LIN {X 0,Y 467.683,Z 145.229,A -85,B 0,C 180,E1 -7462.66,E2 -7462.66} C_VEL
LIN {X 0,Y 467.713,Z 145.224,A -85,B 0,C 180,E1 -7464.827,E2 -7464.827} C_VEL
LIN {X 0,Y 467.852,Z 145.203,A -85,B 0,C 180,E1 -7467.417,E2 -7467.417} C_VEL
LIN {X 0,Y 467.855,Z 145.206,A -85,B 0,C 180,E1 -7470,E2 -7470} C_VEL
LIN {X 0,Y 467.817,Z 145.212,A -85,B 0,C 180,E1 -7472.583,E2 -7472.583} C_VEL
LIN {X 0,Y 467.706,Z 145.226,A -85,B 0,C 180,E1 -7476.038,E2 -7476.038} C_VEL
LIN {X 0,Y 467.661,Z 145.229,A -85,B 0,C 180,E1 -7478.643,E2 -7478.643} C_VEL
LIN {X 0,Y 467.66,Z 145.234,A -85,B 0,C 180,E1 -7482.145,E2 -7482.145} C_VEL
LIN {X 0,Y 467.615,Z 145.236,A -85,B 0,C 180,E1 -7485.696,E2 -7485.696} C_VEL
LIN {X 0,Y 467.621,Z 145.233,A -85,B 0,C 180,E1 -7489.308,E2 -7489.308} C_VEL
LIN {X 0,Y 467.536,Z 145.247,A -85,B 0,C 180,E1 -7492.074,E2 -7492.074} C_VEL
LIN {X 0,Y 467.562,Z 145.239,A -85,B 0,C 180,E1 -7494.89,E2 -7494.89} C_VEL
LIN {X 0,Y 467.548,Z 145.248,A -85,B 0,C 180,E1 -7497.774,E2 -7497.774} C_VEL
LIN {X 0,Y 467.568,Z 145.24,A -85,B 0,C 180,E1 -7501.044,E2 -7501.044} C_VEL
LIN {X 0,Y 467.579,Z 145.238,A -85,B 0,C 180,E1 -7504.24,E2 -7504.24} C_VEL
LIN {X 0,Y 467.545,Z 145.245,A -85,B 0,C 180,E1 -7507.185,E2 -7507.185} C_VEL
LIN {X 0,Y 467.56,Z 145.239,A -85,B 0,C 180,E1 -7510.267,E2 -7510.267} C_VEL
LIN {X 0,Y 467.547,Z 145.243,A -85,B 0,C 180,E1 -7513.746,E2 -7513.746} C_VEL
LIN {X 0,Y 467.547,Z 145.241,A -85,B 0,C 180,E1 -7516.254,E2 -7516.254} C_VEL
LIN {X 0,Y 467.56,Z 145.241,A -85,B 0,C 180,E1 -7519.733,E2 -7519.733} C_VEL
LIN {X 0,Y 467.546,Z 145.245,A -85,B 0,C 180,E1 -7522.815,E2 -7522.815} C_VEL
LIN {X 0,Y 467.579,Z 145.237,A -85,B 0,C 180,E1 -7525.76,E2 -7525.76} C_VEL
LIN {X 0,Y 467.546,Z 145.249,A -85,B 0,C 180,E1 -7528.961,E2 -7528.961} C_VEL
LIN {X 0,Y 467.563,Z 145.24,A -85,B 0,C 180,E1 -7532.227,E2 -7532.227} C_VEL
LIN {X 0,Y 467.563,Z 145.243,A -85,B 0,C 180,E1 -7535.11,E2 -7535.11} C_VEL
LIN {X 0,Y 467.529,Z 145.243,A -85,B 0,C 180,E1 -7537.926,E2 -7537.926} C_VEL
LIN {X 0,Y 467.62,Z 145.24,A -85,B 0,C 180,E1 -7540.692,E2 -7540.692} C_VEL
LIN {X 0,Y 467.616,Z 145.237,A -85,B 0,C 180,E1 -7544.304,E2 -7544.304} C_VEL
LIN {X 0,Y 467.661,Z 145.228,A -85,B 0,C 180,E1 -7547.855,E2 -7547.855} C_VEL
LIN {X 0,Y 467.639,Z 145.229,A -85,B 0,C 180,E1 -7551.356,E2 -7551.356} C_VEL
LIN {X 0,Y 467.705,Z 145.224,A -85,B 0,C 180,E1 -7553.962,E2 -7553.962} C_VEL
LIN {X 0,Y 467.816,Z 145.207,A -85,B 0,C 180,E1 -7557.417,E2 -7557.417} C_VEL
LIN {X 0,Y 467.853,Z 145.208,A -85,B 0,C 180,E1 -7560,E2 -7560} C_VEL
LIN {X 0,Y 467.815,Z 145.21,A -85,B 0,C 180,E1 -7562.583,E2 -7562.583} C_VEL
LIN {X 0,Y 467.704,Z 145.23,A -85,B 0,C 180,E1 -7566.038,E2 -7566.038} C_VEL
LIN {X 0,Y 467.637,Z 145.23,A -85,B 0,C 180,E1 -7568.644,E2 -7568.644} C_VEL
LIN {X 0,Y 467.652,Z 145.23,A -85,B 0,C 180,E1 -7572.354,E2 -7572.354} C_VEL
LIN {X 0,Y 467.574,Z 145.245,A -85,B 0,C 180,E1 -7575.851,E2 -7575.851} C_VEL
LIN {X 0,Y 467.571,Z 145.238,A -85,B 0,C 180,E1 -7578.746,E2 -7578.746} C_VEL
LIN {X 0,Y 467.521,Z 145.247,A -85,B 0,C 180,E1 -7582.075,E2 -7582.075} C_VEL
LIN {X 0,Y 467.553,Z 145.241,A -85,B 0,C 180,E1 -7584.89,E2 -7584.89} C_VEL
LIN {X 0,Y 467.54,Z 145.246,A -85,B 0,C 180,E1 -7587.774,E2 -7587.774} C_VEL
LIN {X 0,Y 467.53,Z 145.246,A -85,B 0,C 180,E1 -7591.036,E2 -7591.036} C_VEL
LIN {X 0,Y 467.567,Z 145.238,A -85,B 0,C 180,E1 -7594.237,E2 -7594.237} C_VEL
LIN {X 0,Y 467.516,Z 145.251,A -85,B 0,C 180,E1 -7597.18,E2 -7597.18} C_VEL
LIN {X 0,Y 467.553,Z 145.24,A -85,B 0,C 180,E1 -7600.267,E2 -7600.267} C_VEL
LIN {X 0,Y 467.519,Z 145.246,A -85,B 0,C 180,E1 -7602.568,E2 -7602.568} C_VEL
LIN {X 0,Y 467.564,Z 145.246,A -85,B 0,C 180,E1 -7605.052,E2 -7605.052} C_VEL
LIN {X 0,Y 467.556,Z 145.244,A -85,B 0,C 180,E1 -7608.727,E2 -7608.727} C_VEL
LIN {X 0,Y 467.539,Z 145.242,A -85,B 0,C 180,E1 -7611.953,E2 -7611.953} C_VEL
LIN {X 0,Y 467.542,Z 145.245,A -85,B 0,C 180,E1 -7615.165,E2 -7615.165} C_VEL
LIN {X 0,Y 467.544,Z 145.243,A -85,B 0,C 180,E1 -7618.257,E2 -7618.257} C_VEL
LIN {X 0,Y 467.526,Z 145.248,A -85,B 0,C 180,E1 -7621.247,E2 -7621.247} C_VEL
LIN {X 0,Y 467.561,Z 145.405,A -85,B 0,C 180,E1 -7624.405,E2 -7624.405} C_VEL
LIN {X 0,Y 469.547,Z 155.588,A -85,B 0,C 180,E1 -7626.398,E2 -7626.398} C_VEL
LIN {X 0,Y 469.65,Z 160.677,A -85,B 0,C 180,E1 -7627.335,E2 -7627.335} C_VEL
LIN {X 0,Y 468.851,Z 179.686,A -85,B 0,C 180,E1 -7630.745,E2 -7630.745} C_VEL
LIN {X 0,Y 468.323,Z 192.549,A -85,B 0,C 180,E1 -7633.009,E2 -7633.009} C_VEL
LIN {X 0,Y 471.154,Z 211.602,A -85,B 0,C 180,E1 -7633.413,E2 -7633.413} C_VEL
LIN {X 0,Y 470.437,Z 300.664,A -85,B 0,C 180,E1 -7634.817,E2 -7634.817} C_VEL
LIN {X 0,Y 470.098,Z 313.865,A -85,B 0,C 180,E1 -7635.194,E2 -7635.194} C_VEL
LIN {X 0,Y 469.617,Z 327.128,A -85,B 0,C 180,E1 -7635.759,E2 -7635.759} C_VEL
LIN {X 0,Y 469.107,Z 339.07,A -85,B 0,C 180,E1 -7636.462,E2 -7636.462} C_VEL
LIN {X 0,Y 468.56,Z 351.287,A -85,B 0,C 180,E1 -7637.392,E2 -7637.392} C_VEL
LIN {X 0,Y 468.159,Z 360.871,A -85,B 0,C 180,E1 -7638.307,E2 -7638.307} C_VEL
LIN {X 0,Y 467.696,Z 370.148,A -85,B 0,C 180,E1 -7639.392,E2 -7639.392} C_VEL
LIN {X 0,Y 467.304,Z 379.162,A -85,B 0,C 180,E1 -7640.696,E2 -7640.696} C_VEL
LIN {X 0,Y 467.007,Z 386.421,A -85,B 0,C 180,E1 -7641.998,E2 -7641.998} C_VEL
LIN {X 0,Y 466.833,Z 391.319,A -85,B 0,C 180,E1 -7643.083,E2 -7643.083} C_VEL
LIN {X 0,Y 466.755,Z 396.078,A -85,B 0,C 180,E1 -7644.383,E2 -7644.383} C_VEL
LIN {X 0,Y 466.645,Z 399.712,A -85,B 0,C 180,E1 -7645.681,E2 -7645.681} C_VEL
LIN {X 0,Y 466.688,Z 401.59,A -85,B 0,C 180,E1 -7646.547,E2 -7646.547} C_VEL
LIN {X 0,Y 466.662,Z 402.997,A -85,B 0,C 180,E1 -7647.41,E2 -7647.41} C_VEL
LIN {X 0,Y 466.62,Z 404.607,A -85,B 0,C 180,E1 -7649.137,E2 -7649.137} C_VEL
LIN {X 0,Y 466.601,Z 404.824,A -85,B 0,C 180,E1 -7650,E2 -7650} C_VEL
LIN {X 0,Y 466.62,Z 404.607,A -85,B 0,C 180,E1 -7650.863,E2 -7650.863} C_VEL
LIN {X 0,Y 466.662,Z 402.991,A -85,B 0,C 180,E1 -7652.59,E2 -7652.59} C_VEL
LIN {X 0,Y 466.688,Z 401.586,A -85,B 0,C 180,E1 -7653.453,E2 -7653.453} C_VEL
LIN {X 0,Y 466.687,Z 398.63,A -85,B 0,C 180,E1 -7654.751,E2 -7654.751} C_VEL
LIN {X 0,Y 466.744,Z 394.631,A -85,B 0,C 180,E1 -7656.05,E2 -7656.05} C_VEL
LIN {X 0,Y 466.94,Z 388.484,A -85,B 0,C 180,E1 -7657.568,E2 -7657.568} C_VEL
LIN {X 0,Y 467.199,Z 381.769,A -85,B 0,C 180,E1 -7658.87,E2 -7658.87} C_VEL
LIN {X 0,Y 467.53,Z 373.439,A -85,B 0,C 180,E1 -7660.174,E2 -7660.174} C_VEL
LIN {X 0,Y 467.998,Z 364.898,A -85,B 0,C 180,E1 -7661.258,E2 -7661.258} C_VEL
LIN {X 0,Y 468.486,Z 354.809,A -85,B 0,C 180,E1 -7662.301,E2 -7662.301} C_VEL
LIN {X 0,Y 468.939,Z 343.914,A -85,B 0,C 180,E1 -7663.212,E2 -7663.212} C_VEL
LIN {X 0,Y 469.412,Z 332.466,A -85,B 0,C 180,E1 -7663.971,E2 -7663.971} C_VEL
LIN {X 0,Y 469.895,Z 320.661,A -85,B 0,C 180,E1 -7664.564,E2 -7664.564} C_VEL
LIN {X 0,Y 470.317,Z 307.075,A -85,B 0,C 180,E1 -7665.049,E2 -7665.049} C_VEL
LIN {X 0,Y 470.645,Z 293.364,A -85,B 0,C 180,E1 -7665.343,E2 -7665.343} C_VEL
LIN {X 0,Y 471.151,Z 210.06,A -85,B 0,C 180,E1 -7666.648,E2 -7666.648} C_VEL
LIN {X 0,Y 468.307,Z 191.951,A -85,B 0,C 180,E1 -7667.066,E2 -7667.066} C_VEL
LIN {X 0,Y 468.86,Z 176.916,A -85,B 0,C 180,E1 -7669.711,E2 -7669.711} C_VEL
LIN {X 0,Y 469.689,Z 159.022,A -85,B 0,C 180,E1 -7672.895,E2 -7672.895} C_VEL
LIN {X 0,Y 469.27,Z 153.888,A -85,B 0,C 180,E1 -7673.852,E2 -7673.852} C_VEL
LIN {X 0,Y 467.557,Z 145.248,A -85,B 0,C 180,E1 -7675.544,E2 -7675.544} C_VEL
LIN {X 0,Y 467.526,Z 145.25,A -85,B 0,C 180,E1 -7678.753,E2 -7678.753} C_VEL
LIN {X 0,Y 467.544,Z 145.249,A -85,B 0,C 180,E1 -7681.743,E2 -7681.743} C_VEL
LIN {X 0,Y 467.541,Z 145.248,A -85,B 0,C 180,E1 -7684.835,E2 -7684.835} C_VEL
LIN {X 0,Y 467.535,Z 145.244,A -85,B 0,C 180,E1 -7688.048,E2 -7688.048} C_VEL
LIN {X 0,Y 467.551,Z 145.245,A -85,B 0,C 180,E1 -7691.406,E2 -7691.406} C_VEL
LIN {X 0,Y 467.564,Z 145.247,A -85,B 0,C 180,E1 -7695.052,E2 -7695.052} C_VEL
LIN {X 0,Y 467.552,Z 145.246,A -85,B 0,C 180,E1 -7698.728,E2 -7698.728} C_VEL
LIN {X 0,Y 467.536,Z 145.243,A -85,B 0,C 180,E1 -7701.953,E2 -7701.953} C_VEL
LIN {X 0,Y 467.543,Z 145.245,A -85,B 0,C 180,E1 -7705.165,E2 -7705.165} C_VEL
LIN {X 0,Y 467.545,Z 145.242,A -85,B 0,C 180,E1 -7708.257,E2 -7708.257} C_VEL
LIN {X 0,Y 467.527,Z 145.243,A -85,B 0,C 180,E1 -7711.247,E2 -7711.247} C_VEL
LIN {X 0,Y 467.564,Z 145.243,A -85,B 0,C 180,E1 -7714.406,E2 -7714.406} C_VEL
LIN {X 0,Y 467.549,Z 145.244,A -85,B 0,C 180,E1 -7716.994,E2 -7716.994} C_VEL
LIN {X 0,Y 467.541,Z 145.237,A -85,B 0,C 180,E1 -7719.773,E2 -7719.773} C_VEL
LIN {X 0,Y 467.555,Z 145.246,A -85,B 0,C 180,E1 -7722.505,E2 -7722.505} C_VEL
LIN {X 0,Y 467.562,Z 145.238,A -85,B 0,C 180,E1 -7725.195,E2 -7725.195} C_VEL
LIN {X 0,Y 467.645,Z 145.23,A -85,B 0,C 180,E1 -7727.854,E2 -7727.854} C_VEL
LIN {X 0,Y 467.633,Z 145.23,A -85,B 0,C 180,E1 -7731.356,E2 -7731.356} C_VEL
LIN {X 0,Y 467.697,Z 145.221,A -85,B 0,C 180,E1 -7733.962,E2 -7733.962} C_VEL
LIN {X 0,Y 467.815,Z 145.205,A -85,B 0,C 180,E1 -7737.417,E2 -7737.417} C_VEL
LIN {X 0,Y 467.853,Z 145.208,A -85,B 0,C 180,E1 -7740,E2 -7740} C_VEL
LIN {X 0,Y 467.815,Z 145.209,A -85,B 0,C 180,E1 -7742.583,E2 -7742.583} C_VEL
LIN {X 0,Y 467.704,Z 145.225,A -85,B 0,C 180,E1 -7746.038,E2 -7746.038} C_VEL
LIN {X 0,Y 467.637,Z 145.23,A -85,B 0,C 180,E1 -7748.644,E2 -7748.644} C_VEL
LIN {X 0,Y 467.652,Z 145.231,A -85,B 0,C 180,E1 -7752.146,E2 -7752.146} C_VEL
LIN {X 0,Y 467.617,Z 145.237,A -85,B 0,C 180,E1 -7755.696,E2 -7755.696} C_VEL
LIN {X 0,Y 467.576,Z 145.238,A -85,B 0,C 180,E1 -7758.748,E2 -7758.748} C_VEL
LIN {X 0,Y 467.562,Z 145.242,A -85,B 0,C 180,E1 -7761.261,E2 -7761.261} C_VEL
LIN {X 0,Y 467.558,Z 145.246,A -85,B 0,C 180,E1 -7763.944,E2 -7763.944} C_VEL
LIN {X 0,Y 467.538,Z 145.246,A -85,B 0,C 180,E1 -7766.805,E2 -7766.805} C_VEL
LIN {X 0,Y 467.538,Z 145.249,A -85,B 0,C 180,E1 -7769.739,E2 -7769.739} C_VEL
LIN {X 0,Y 467.577,Z 145.242,A -85,B 0,C 180,E1 -7772.759,E2 -7772.759} C_VEL
LIN {X 0,Y 467.567,Z 145.246,A -85,B 0,C 180,E1 -7775.889,E2 -7775.889} C_VEL
LIN {X 0,Y 467.613,Z 145.348,A -85,B 0,C 180,E1 -7776.318,E2 -7776.318} C_VEL
LIN {X 0,Y 468.909,Z 152.961,A -85,B 0,C 180,E1 -7777.916,E2 -7777.916} C_VEL
LIN {X 0,Y 468.662,Z 165.61,A -85,B 0,C 180,E1 -7780.434,E2 -7780.434} C_VEL
LIN {X 0,Y 468.541,Z 168.542,A -85,B 0,C 180,E1 -7781.014,E2 -7781.014} C_VEL
LIN {X 0,Y 471.427,Z 183.586,A -85,B 0,C 180,E1 -7781.373,E2 -7781.373} C_VEL
LIN {X 0,Y 470.577,Z 276.466,A -85,B 0,C 180,E1 -7782.849,E2 -7782.849} C_VEL
LIN {X 0,Y 470.298,Z 290.13,A -85,B 0,C 180,E1 -7783.255,E2 -7783.255} C_VEL
LIN {X 0,Y 469.95,Z 302.218,A -85,B 0,C 180,E1 -7783.785,E2 -7783.785} C_VEL
LIN {X 0,Y 469.476,Z 313.638,A -85,B 0,C 180,E1 -7784.456,E2 -7784.456} C_VEL
LIN {X 0,Y 468.981,Z 325.331,A -85,B 0,C 180,E1 -7785.343,E2 -7785.343} C_VEL
LIN {X 0,Y 468.475,Z 336.021,A -85,B 0,C 180,E1 -7786.363,E2 -7786.363} C_VEL
LIN {X 0,Y 467.997,Z 345.447,A -85,B 0,C 180,E1 -7787.485,E2 -7787.485} C_VEL
LIN {X 0,Y 467.583,Z 353.89,A -85,B 0,C 180,E1 -7788.723,E2 -7788.723} C_VEL
LIN {X 0,Y 467.232,Z 361.432,A -85,B 0,C 180,E1 -7790.097,E2 -7790.097} C_VEL
LIN {X 0,Y 466.981,Z 367.45,A -85,B 0,C 180,E1 -7791.499,E2 -7791.499} C_VEL
LIN {X 0,Y 466.806,Z 372.297,A -85,B 0,C 180,E1 -7792.971,E2 -7792.971} C_VEL
LIN {X 0,Y 466.634,Z 375.76,A -85,B 0,C 180,E1 -7794.42,E2 -7794.42} C_VEL
LIN {X 0,Y 466.534,Z 378.282,A -85,B 0,C 180,E1 -7796.125,E2 -7796.125} C_VEL
LIN {X 0,Y 466.51,Z 379.06,A -85,B 0,C 180,E1 -7797.217,E2 -7797.217} C_VEL
LIN {X 0,Y 465.851,Z 379.263,A -85,B 0,C 180,E1 -7797.938,E2 -7797.938} C_VEL
LIN {X 0,Y 463.014,Z 379.028,A -85,B 0,C 180,E1 -7799.111,E2 -7799.111} C_VEL
LIN {X 0,Y 460.619,Z 378.334,A -85,B 0,C 180,E1 -7800.053,E2 -7800.053} C_VEL
LIN {X 0,Y 459.537,Z 377.298,A -85,B 0,C 180,E1 -7800.894,E2 -7800.894} C_VEL
LIN {X 0,Y 459.517,Z 377.041,A -85,B 0,C 180,E1 -7801.015,E2 -7801.015} C_VEL
LIN {X 0,Y 459.644,Z 374.212,A -85,B 0,C 180,E1 -7802.478,E2 -7802.478} C_VEL
LIN {X 0,Y 459.894,Z 369.669,A -85,B 0,C 180,E1 -7804.067,E2 -7804.067} C_VEL
LIN {X 0,Y 460.064,Z 363.549,A -85,B 0,C 180,E1 -7805.641,E2 -7805.641} C_VEL
LIN {X 0,Y 460.415,Z 356.212,A -85,B 0,C 180,E1 -7807.092,E2 -7807.092} C_VEL
LIN {X 0,Y 460.81,Z 348.502,A -85,B 0,C 180,E1 -7808.317,E2 -7808.317} C_VEL
LIN {X 0,Y 461.276,Z 339.442,A -85,B 0,C 180,E1 -7809.486,E2 -7809.486} C_VEL
LIN {X 0,Y 461.796,Z 328.795,A -85,B 0,C 180,E1 -7810.592,E2 -7810.592} C_VEL
LIN {X 0,Y 462.388,Z 317.849,A -85,B 0,C 180,E1 -7811.501,E2 -7811.501} C_VEL
LIN {X 0,Y 462.805,Z 306.173,A -85,B 0,C 180,E1 -7812.262,E2 -7812.262} C_VEL
LIN {X 0,Y 463.234,Z 292.993,A -85,B 0,C 180,E1 -7812.904,E2 -7812.904} C_VEL
LIN {X 0,Y 463.559,Z 280.962,A -85,B 0,C 180,E1 -7813.315,E2 -7813.315} C_VEL
LIN {X 0,Y 463.764,Z 266.671,A -85,B 0,C 180,E1 -7813.605,E2 -7813.605} C_VEL
LIN {X 0,Y 464.504,Z 184.737,A -85,B 0,C 180,E1 -7814.899,E2 -7814.899} C_VEL
LIN {X 0,Y 461.504,Z 168.599,A -85,B 0,C 180,E1 -7815.278,E2 -7815.278} C_VEL
LIN {X 0,Y 461.992,Z 154.759,A -85,B 0,C 180,E1 -7818.149,E2 -7818.149} C_VEL
LIN {X 0,Y 460.626,Z 146.11,A -85,B 0,C 180,E1 -7820.061,E2 -7820.061} C_VEL
LIN {X 0,Y 460.612,Z 146.111,A -85,B 0,C 180,E1 -7822.989,E2 -7822.989} C_VEL
LIN {X 0,Y 460.685,Z 146.1,A -85,B 0,C 180,E1 -7824.748,E2 -7824.748} C_VEL
LIN {X 0,Y 460.792,Z 146.082,A -85,B 0,C 180,E1 -7827.377,E2 -7827.377} C_VEL
LIN {X 0,Y 460.825,Z 146.081,A -85,B 0,C 180,E1 -7830,E2 -7830} C_VEL
LIN {X 0,Y 460.761,Z 146.09,A -85,B 0,C 180,E1 -7832.623,E2 -7832.623} C_VEL
LIN {X 0,Y 460.672,Z 146.104,A -85,B 0,C 180,E1 -7836.13,E2 -7836.13} C_VEL
LIN {X 0,Y 460.613,Z 146.106,A -85,B 0,C 180,E1 -7838.776,E2 -7838.776} C_VEL
LIN {X 0,Y 460.612,Z 146.109,A -85,B 0,C 180,E1 -7842.334,E2 -7842.334} C_VEL
LIN {X 0,Y 460.559,Z 146.119,A -85,B 0,C 180,E1 -7845.978,E2 -7845.978} C_VEL
LIN {X 0,Y 460.568,Z 146.114,A -85,B 0,C 180,E1 -7849.616,E2 -7849.616} C_VEL
LIN {X 0,Y 460.513,Z 146.118,A -85,B 0,C 180,E1 -7852.429,E2 -7852.429} C_VEL
LIN {X 0,Y 460.537,Z 146.122,A -85,B 0,C 180,E1 -7855.793,E2 -7855.793} C_VEL
LIN {X 0,Y 460.523,Z 146.118,A -85,B 0,C 180,E1 -7859.232,E2 -7859.232} C_VEL
LIN {X 0,Y 460.528,Z 146.116,A -85,B 0,C 180,E1 -7862.285,E2 -7862.285} C_VEL
LIN {X 0,Y 460.509,Z 146.125,A -85,B 0,C 180,E1 -7865.446,E2 -7865.446} C_VEL
LIN {X 0,Y 460.507,Z 146.12,A -85,B 0,C 180,E1 -7868.891,E2 -7868.891} C_VEL
LIN {X 0,Y 460.505,Z 146.123,A -85,B 0,C 180,E1 -7871.598,E2 -7871.598} C_VEL
LIN {X 0,Y 460.514,Z 146.118,A -85,B 0,C 180,E1 -7874.589,E2 -7874.589} C_VEL
LIN {X 0,Y 460.478,Z 146.123,A -85,B 0,C 180,E1 -7877.813,E2 -7877.813} C_VEL
LIN {X 0,Y 460.516,Z 146.117,A -85,B 0,C 180,E1 -7880.136,E2 -7880.136} C_VEL
LIN {X 0,Y 460.476,Z 146.125,A -85,B 0,C 180,E1 -7883.47,E2 -7883.47} C_VEL
LIN {X 0,Y 460.519,Z 146.12,A -85,B 0,C 180,E1 -7886.674,E2 -7886.674} C_VEL
LIN {X 0,Y 460.5,Z 146.119,A -85,B 0,C 180,E1 -7889.759,E2 -7889.759} C_VEL
LIN {X 0,Y 460.516,Z 146.123,A -85,B 0,C 180,E1 -7892.752,E2 -7892.752} C_VEL
LIN {X 0,Y 460.521,Z 146.116,A -85,B 0,C 180,E1 -7895.666,E2 -7895.666} C_VEL
LIN {X 0,Y 460.522,Z 146.122,A -85,B 0,C 180,E1 -7898.58,E2 -7898.58} C_VEL
LIN {X 0,Y 460.586,Z 146.109,A -85,B 0,C 180,E1 -7901.311,E2 -7901.311} C_VEL
LIN {X 0,Y 460.549,Z 146.115,A -85,B 0,C 180,E1 -7904.964,E2 -7904.964} C_VEL
LIN {X 0,Y 460.613,Z 146.111,A -85,B 0,C 180,E1 -7908.559,E2 -7908.559} C_VEL
LIN {X 0,Y 460.597,Z 146.107,A -85,B 0,C 180,E1 -7911.223,E2 -7911.223} C_VEL
LIN {X 0,Y 460.671,Z 146.1,A -85,B 0,C 180,E1 -7913.87,E2 -7913.87} C_VEL
LIN {X 0,Y 460.76,Z 146.086,A -85,B 0,C 180,E1 -7917.377,E2 -7917.377} C_VEL
LIN {X 0,Y 460.823,Z 146.084,A -85,B 0,C 180,E1 -7920,E2 -7920} C_VEL
LIN {X 0,Y 460.759,Z 146.088,A -85,B 0,C 180,E1 -7922.623,E2 -7922.623} C_VEL
LIN {X 0,Y 460.67,Z 146.104,A -85,B 0,C 180,E1 -7926.13,E2 -7926.13} C_VEL
LIN {X 0,Y 460.592,Z 146.108,A -85,B 0,C 180,E1 -7928.777,E2 -7928.777} C_VEL
LIN {X 0,Y 460.601,Z 146.108,A -85,B 0,C 180,E1 -7932.435,E2 -7932.435} C_VEL
LIN {X 0,Y 460.529,Z 146.121,A -85,B 0,C 180,E1 -7935.964,E2 -7935.964} C_VEL
LIN {X 0,Y 460.53,Z 146.115,A -85,B 0,C 180,E1 -7938.885,E2 -7938.885} C_VEL
LIN {X 0,Y 460.495,Z 146.12,A -85,B 0,C 180,E1 -7942.43,E2 -7942.43} C_VEL
LIN {X 0,Y 460.524,Z 146.121,A -85,B 0,C 180,E1 -7945.789,E2 -7945.789} C_VEL
LIN {X 0,Y 460.498,Z 146.119,A -85,B 0,C 180,E1 -7948.237,E2 -7948.237} C_VEL
LIN {X 0,Y 460.498,Z 146.125,A -85,B 0,C 180,E1 -7951.277,E2 -7951.277} C_VEL
LIN {X 0,Y 460.513,Z 146.117,A -85,B 0,C 180,E1 -7954.501,E2 -7954.501} C_VEL
LIN {X 0,Y 460.483,Z 146.124,A -85,B 0,C 180,E1 -7957.625,E2 -7957.625} C_VEL
LIN {X 0,Y 460.515,Z 146.122,A -85,B 0,C 180,E1 -7961.013,E2 -7961.013} C_VEL
LIN {X 0,Y 460.512,Z 146.119,A -85,B 0,C 180,E1 -7964.589,E2 -7964.589} C_VEL
LIN {X 0,Y 460.474,Z 146.122,A -85,B 0,C 180,E1 -7967.813,E2 -7967.813} C_VEL
LIN {X 0,Y 460.497,Z 146.119,A -85,B 0,C 180,E1 -7970.134,E2 -7970.134} C_VEL
LIN {X 0,Y 460.458,Z 146.125,A -85,B 0,C 180,E1 -7973.469,E2 -7973.469} C_VEL
LIN {X 0,Y 460.501,Z 146.125,A -85,B 0,C 180,E1 -7976.673,E2 -7976.673} C_VEL
LIN {X 0,Y 460.479,Z 146.124,A -85,B 0,C 180,E1 -7979.757,E2 -7979.757} C_VEL
LIN {X 0,Y 460.485,Z 146.128,A -85,B 0,C 180,E1 -7982.75,E2 -7982.75} C_VEL
LIN {X 0,Y 460.546,Z 146.304,A -85,B 0,C 180,E1 -7984.204,E2 -7984.204} C_VEL
LIN {X 0,Y 462.709,Z 157.916,A -85,B 0,C 180,E1 -7986.504,E2 -7986.504} C_VEL
LIN {X 0,Y 462.351,Z 169.326,A -85,B 0,C 180,E1 -7988.604,E2 -7988.604} C_VEL
LIN {X 0,Y 461.645,Z 184.525,A -85,B 0,C 180,E1 -7991.355,E2 -7991.355} C_VEL
LIN {X 0,Y 461.351,Z 192.266,A -85,B 0,C 180,E1 -7992.746,E2 -7992.746} C_VEL
LIN {X 0,Y 464.335,Z 211.934,A -85,B 0,C 180,E1 -7993.178,E2 -7993.178} C_VEL
LIN {X 0,Y 463.596,Z 300.067,A -85,B 0,C 180,E1 -7994.587,E2 -7994.587} C_VEL
LIN {X 0,Y 463.226,Z 313.409,A -85,B 0,C 180,E1 -7994.969,E2 -7994.969} C_VEL
LIN {X 0,Y 462.738,Z 326.75,A -85,B 0,C 180,E1 -7995.543,E2 -7995.543} C_VEL
LIN {X 0,Y 462.181,Z 338.745,A -85,B 0,C 180,E1 -7996.255,E2 -7996.255} C_VEL
LIN {X 0,Y 461.65,Z 350.343,A -85,B 0,C 180,E1 -7997.145,E2 -7997.145} C_VEL
LIN {X 0,Y 461.19,Z 360.599,A -85,B 0,C 180,E1 -7998.128,E2 -7998.128} C_VEL
LIN {X 0,Y 460.662,Z 369.896,A -85,B 0,C 180,E1 -7999.229,E2 -7999.229} C_VEL
LIN {X 0,Y 460.258,Z 378.924,A -85,B 0,C 180,E1 -8000.552,E2 -8000.552} C_VEL
LIN {X 0,Y 459.948,Z 386.193,A -85,B 0,C 180,E1 -8001.875,E2 -8001.875} C_VEL
LIN {X 0,Y 459.737,Z 392.286,A -85,B 0,C 180,E1 -8003.272,E2 -8003.272} C_VEL
LIN {X 0,Y 459.647,Z 397.193,A -85,B 0,C 180,E1 -8004.736,E2 -8004.736} C_VEL
LIN {X 0,Y 459.563,Z 399.505,A -85,B 0,C 180,E1 -8005.615,E2 -8005.615} C_VEL
LIN {X 0,Y 459.583,Z 401.385,A -85,B 0,C 180,E1 -8006.493,E2 -8006.493} C_VEL
LIN {X 0,Y 459.584,Z 402.797,A -85,B 0,C 180,E1 -8007.371,E2 -8007.371} C_VEL
LIN {X 0,Y 459.523,Z 404.41,A -85,B 0,C 180,E1 -8009.124,E2 -8009.124} C_VEL
LIN {X 0,Y 459.533,Z 404.63,A -85,B 0,C 180,E1 -8010,E2 -8010} C_VEL
LIN {X 0,Y 459.523,Z 404.414,A -85,B 0,C 180,E1 -8010.876,E2 -8010.876} C_VEL
LIN {X 0,Y 459.584,Z 402.8,A -85,B 0,C 180,E1 -8012.629,E2 -8012.629} C_VEL
LIN {X 0,Y 459.583,Z 401.395,A -85,B 0,C 180,E1 -8013.507,E2 -8013.507} C_VEL
LIN {X 0,Y 459.615,Z 398.44,A -85,B 0,C 180,E1 -8014.824,E2 -8014.824} C_VEL
LIN {X 0,Y 459.714,Z 393.408,A -85,B 0,C 180,E1 -8016.431,E2 -8016.431} C_VEL
LIN {X 0,Y 459.898,Z 387.282,A -85,B 0,C 180,E1 -8017.905,E2 -8017.905} C_VEL
LIN {X 0,Y 460.196,Z 380.345,A -85,B 0,C 180,E1 -8019.228,E2 -8019.228} C_VEL
LIN {X 0,Y 460.488,Z 373.262,A -85,B 0,C 180,E1 -8020.331,E2 -8020.331} C_VEL
LIN {X 0,Y 461.016,Z 364.728,A -85,B 0,C 180,E1 -8021.431,E2 -8021.431} C_VEL
LIN {X 0,Y 461.504,Z 354.852,A -85,B 0,C 180,E1 -8022.47,E2 -8022.47} C_VEL
LIN {X 0,Y 462.016,Z 343.755,A -85,B 0,C 180,E1 -8023.414,E2 -8023.414} C_VEL
LIN {X 0,Y 462.525,Z 332.32,A -85,B 0,C 180,E1 -8024.183,E2 -8024.183} C_VEL
LIN {X 0,Y 463.033,Z 320.547,A -85,B 0,C 180,E1 -8024.785,E2 -8024.785} C_VEL
LIN {X 0,Y 463.485,Z 307.01,A -85,B 0,C 180,E1 -8025.276,E2 -8025.276} C_VEL
LIN {X 0,Y 463.826,Z 293.453,A -85,B 0,C 180,E1 -8025.574,E2 -8025.574} C_VEL
LIN {X 0,Y 464.322,Z 210.557,A -85,B 0,C 180,E1 -8026.897,E2 -8026.897} C_VEL
LIN {X 0,Y 461.359,Z 191.816,A -85,B 0,C 180,E1 -8027.326,E2 -8027.326} C_VEL
LIN {X 0,Y 462.014,Z 175.48,A -85,B 0,C 180,E1 -8030.247,E2 -8030.247} C_VEL
LIN {X 0,Y 462.772,Z 158.873,A -85,B 0,C 180,E1 -8033.257,E2 -8033.257} C_VEL
LIN {X 0,Y 461.291,Z 149.874,A -85,B 0,C 180,E1 -8035.011,E2 -8035.011} C_VEL
LIN {X 0,Y 460.524,Z 146.122,A -85,B 0,C 180,E1 -8035.79,E2 -8035.79} C_VEL
LIN {X 0,Y 460.497,Z 146.125,A -85,B 0,C 180,E1 -8038.237,E2 -8038.237} C_VEL
LIN {X 0,Y 460.497,Z 146.129,A -85,B 0,C 180,E1 -8041.278,E2 -8041.278} C_VEL
LIN {X 0,Y 460.51,Z 146.122,A -85,B 0,C 180,E1 -8044.501,E2 -8044.501} C_VEL
LIN {X 0,Y 460.479,Z 146.125,A -85,B 0,C 180,E1 -8047.626,E2 -8047.626} C_VEL
LIN {X 0,Y 460.501,Z 146.128,A -85,B 0,C 180,E1 -8051.015,E2 -8051.015} C_VEL
LIN {X 0,Y 460.512,Z 146.122,A -85,B 0,C 180,E1 -8054.59,E2 -8054.59} C_VEL
LIN {X 0,Y 460.473,Z 146.124,A -85,B 0,C 180,E1 -8057.813,E2 -8057.813} C_VEL
LIN {X 0,Y 460.476,Z 146.121,A -85,B 0,C 180,E1 -8060.132,E2 -8060.132} C_VEL
LIN {X 0,Y 460.457,Z 146.124,A -85,B 0,C 180,E1 -8063.469,E2 -8063.469} C_VEL
LIN {X 0,Y 460.503,Z 146.122,A -85,B 0,C 180,E1 -8066.673,E2 -8066.673} C_VEL
LIN {X 0,Y 460.481,Z 146.121,A -85,B 0,C 180,E1 -8069.758,E2 -8069.758} C_VEL
LIN {X 0,Y 460.487,Z 146.127,A -85,B 0,C 180,E1 -8072.751,E2 -8072.751} C_VEL
LIN {X 0,Y 460.498,Z 146.116,A -85,B 0,C 180,E1 -8075.665,E2 -8075.665} C_VEL
LIN {X 0,Y 460.513,Z 146.12,A -85,B 0,C 180,E1 -8078.583,E2 -8078.583} C_VEL
LIN {X 0,Y 460.53,Z 146.116,A -85,B 0,C 180,E1 -8081.308,E2 -8081.308} C_VEL
LIN {X 0,Y 460.524,Z 146.117,A -85,B 0,C 180,E1 -8084.056,E2 -8084.056} C_VEL
LIN {X 0,Y 460.605,Z 146.106,A -85,B 0,C 180,E1 -8087.666,E2 -8087.666} C_VEL
LIN {X 0,Y 460.589,Z 146.107,A -85,B 0,C 180,E1 -8091.223,E2 -8091.223} C_VEL
LIN {X 0,Y 460.664,Z 146.096,A -85,B 0,C 180,E1 -8093.869,E2 -8093.869} C_VEL
LIN {X 0,Y 460.758,Z 146.084,A -85,B 0,C 180,E1 -8097.377,E2 -8097.377} C_VEL
LIN {X 0,Y 460.822,Z 146.084,A -85,B 0,C 180,E1 -8100,E2 -8100} C_VEL
LIN {X 0,Y 460.759,Z 146.088,A -85,B 0,C 180,E1 -8102.623,E2 -8102.623} C_VEL
LIN {X 0,Y 460.671,Z 146.101,A -85,B 0,C 180,E1 -8106.13,E2 -8106.13} C_VEL
LIN {X 0,Y 460.592,Z 146.107,A -85,B 0,C 180,E1 -8108.777,E2 -8108.777} C_VEL
LIN {X 0,Y 460.601,Z 146.107,A -85,B 0,C 180,E1 -8112.435,E2 -8112.435} C_VEL
LIN {X 0,Y 460.561,Z 146.117,A -85,B 0,C 180,E1 -8115.978,E2 -8115.978} C_VEL
LIN {X 0,Y 460.534,Z 146.115,A -85,B 0,C 180,E1 -8118.886,E2 -8118.886} C_VEL
LIN {X 0,Y 460.513,Z 146.123,A -85,B 0,C 180,E1 -8121.486,E2 -8121.486} C_VEL
LIN {X 0,Y 460.521,Z 146.12,A -85,B 0,C 180,E1 -8124.334,E2 -8124.334} C_VEL
LIN {X 0,Y 460.494,Z 146.127,A -85,B 0,C 180,E1 -8127.249,E2 -8127.249} C_VEL
LIN {X 0,Y 460.5,Z 146.123,A -85,B 0,C 180,E1 -8130.241,E2 -8130.241} C_VEL
LIN {X 0,Y 460.52,Z 146.123,A -85,B 0,C 180,E1 -8133.326,E2 -8133.326} C_VEL
LIN {X 0,Y 460.569,Z 146.269,A -85,B 0,C 180,E1 -8136.121,E2 -8136.121} C_VEL
LIN {X 0,Y 461.919,Z 153.671,A -85,B 0,C 180,E1 -8137.704,E2 -8137.704} C_VEL
LIN {X 0,Y 461.782,Z 163.71,A -85,B 0,C 180,E1 -8139.733,E2 -8139.733} C_VEL
LIN {X 0,Y 461.617,Z 168.827,A -85,B 0,C 180,E1 -8140.746,E2 -8140.746} C_VEL
LIN {X 0,Y 464.59,Z 183.936,A -85,B 0,C 180,E1 -8141.115,E2 -8141.115} C_VEL
LIN {X 0,Y 463.756,Z 276.622,A -85,B 0,C 180,E1 -8142.614,E2 -8142.614} C_VEL
LIN {X 0,Y 463.483,Z 290.022,A -85,B 0,C 180,E1 -8143.016,E2 -8143.016} C_VEL
LIN {X 0,Y 463.097,Z 302.314,A -85,B 0,C 180,E1 -8143.559,E2 -8143.559} C_VEL
LIN {X 0,Y 462.55,Z 314.455,A -85,B 0,C 180,E1 -8144.289,E2 -8144.289} C_VEL
LIN {X 0,Y 462.057,Z 325.458,A -85,B 0,C 180,E1 -8145.14,E2 -8145.14} C_VEL
LIN {X 0,Y 461.531,Z 335.875,A -85,B 0,C 180,E1 -8146.143,E2 -8146.143} C_VEL
LIN {X 0,Y 461.015,Z 345.372,A -85,B 0,C 180,E1 -8147.282,E2 -8147.282} C_VEL
LIN {X 0,Y 460.612,Z 352.934,A -85,B 0,C 180,E1 -8148.387,E2 -8148.387} C_VEL
LIN {X 0,Y 460.271,Z 360.631,A -85,B 0,C 180,E1 -8149.771,E2 -8149.771} C_VEL
LIN {X 0,Y 459.979,Z 366.977,A -85,B 0,C 180,E1 -8151.212,E2 -8151.212} C_VEL
LIN {X 0,Y 459.741,Z 371.82,A -85,B 0,C 180,E1 -8152.648,E2 -8152.648} C_VEL
LIN {X 0,Y 459.6,Z 375.512,A -85,B 0,C 180,E1 -8154.141,E2 -8154.141} C_VEL
LIN {X 0,Y 459.466,Z 378.03,A -85,B 0,C 180,E1 -8155.689,E2 -8155.689} C_VEL
LIN {X 0,Y 459.415,Z 379.312,A -85,B 0,C 180,E1 -8157.286,E2 -8157.286} C_VEL
LIN {X 0,Y 459.438,Z 379.209,A -85,B 0,C 180,E1 -8158.941,E2 -8158.941} C_VEL
LIN {X 0,Y 459.522,Z 377.571,A -85,B 0,C 180,E1 -8160.698,E2 -8160.698} C_VEL
LIN {X 0,Y 459.517,Z 377.041,A -85,B 0,C 180,E1 -8161.015,E2 -8161.015} C_VEL
LIN {X 0,Y 458.878,Z 375.872,A -85,B 0,C 180,E1 -8161.731,E2 -8161.731} C_VEL
LIN {X 0,Y 456.126,Z 373.403,A -85,B 0,C 180,E1 -8162.883,E2 -8162.883} C_VEL
LIN {X 0,Y 453.845,Z 370.936,A -85,B 0,C 180,E1 -8163.795,E2 -8163.795} C_VEL
LIN {X 0,Y 452.932,Z 368.729,A -85,B 0,C 180,E1 -8164.483,E2 -8164.483} C_VEL
LIN {X 0,Y 452.893,Z 367.903,A -85,B 0,C 180,E1 -8164.712,E2 -8164.712} C_VEL
LIN {X 0,Y 453.131,Z 361.622,A -85,B 0,C 180,E1 -8166.218,E2 -8166.218} C_VEL
LIN {X 0,Y 453.509,Z 353.712,A -85,B 0,C 180,E1 -8167.686,E2 -8167.686} C_VEL
LIN {X 0,Y 453.965,Z 345.516,A -85,B 0,C 180,E1 -8168.911,E2 -8168.911} C_VEL
LIN {X 0,Y 454.528,Z 335.579,A -85,B 0,C 180,E1 -8170.113,E2 -8170.113} C_VEL
LIN {X 0,Y 455.067,Z 324.356,A -85,B 0,C 180,E1 -8171.192,E2 -8171.192} C_VEL
LIN {X 0,Y 455.645,Z 313.365,A -85,B 0,C 180,E1 -8172.032,E2 -8172.032} C_VEL
LIN {X 0,Y 456.084,Z 301.174,A -85,B 0,C 180,E1 -8172.754,E2 -8172.754} C_VEL
LIN {X 0,Y 456.519,Z 288.302,A -85,B 0,C 180,E1 -8173.309,E2 -8173.309} C_VEL
LIN {X 0,Y 456.819,Z 276.063,A -85,B 0,C 180,E1 -8173.665,E2 -8173.665} C_VEL
LIN {X 0,Y 457.688,Z 185.177,A -85,B 0,C 180,E1 -8175.145,E2 -8175.145} C_VEL
LIN {X 0,Y 454.564,Z 168.765,A -85,B 0,C 180,E1 -8175.542,E2 -8175.542} C_VEL
LIN {X 0,Y 455.045,Z 156.149,A -85,B 0,C 180,E1 -8178.191,E2 -8178.191} C_VEL
LIN {X 0,Y 453.62,Z 147.201,A -85,B 0,C 180,E1 -8180.187,E2 -8180.187} C_VEL
LIN {X 0,Y 453.577,Z 146.989,A -85,B 0,C 180,E1 -8180.637,E2 -8180.637} C_VEL
LIN {X 0,Y 453.644,Z 146.977,A -85,B 0,C 180,E1 -8183.774,E2 -8183.774} C_VEL
LIN {X 0,Y 453.736,Z 146.961,A -85,B 0,C 180,E1 -8187.337,E2 -8187.337} C_VEL
LIN {X 0,Y 453.794,Z 146.957,A -85,B 0,C 180,E1 -8190,E2 -8190} C_VEL
LIN {X 0,Y 453.708,Z 146.968,A -85,B 0,C 180,E1 -8192.664,E2 -8192.664} C_VEL
LIN {X 0,Y 453.639,Z 146.981,A -85,B 0,C 180,E1 -8196.226,E2 -8196.226} C_VEL
LIN {X 0,Y 453.58,Z 146.981,A -85,B 0,C 180,E1 -8198.914,E2 -8198.914} C_VEL
LIN {X 0,Y 453.567,Z 146.985,A -85,B 0,C 180,E1 -8202.529,E2 -8202.529} C_VEL
LIN {X 0,Y 453.505,Z 146.997,A -85,B 0,C 180,E1 -8206.091,E2 -8206.091} C_VEL
LIN {X 0,Y 453.519,Z 146.988,A -85,B 0,C 180,E1 -8209.039,E2 -8209.039} C_VEL
LIN {X 0,Y 453.479,Z 147.001,A -85,B 0,C 180,E1 -8211.836,E2 -8211.836} C_VEL
LIN {X 0,Y 453.472,Z 146.994,A -85,B 0,C 180,E1 -8214.737,E2 -8214.737} C_VEL
LIN {X 0,Y 453.465,Z 147,A -85,B 0,C 180,E1 -8217.943,E2 -8217.943} C_VEL
LIN {X 0,Y 453.477,Z 146.994,A -85,B 0,C 180,E1 -8220.76,E2 -8220.76} C_VEL
LIN {X 0,Y 453.469,Z 146.998,A -85,B 0,C 180,E1 -8223.914,E2 -8223.914} C_VEL
LIN {X 0,Y 453.452,Z 147.001,A -85,B 0,C 180,E1 -8227.19,E2 -8227.19} C_VEL
LIN {X 0,Y 453.472,Z 146.994,A -85,B 0,C 180,E1 -8230.612,E2 -8230.612} C_VEL
LIN {X 0,Y 453.484,Z 146.993,A -85,B 0,C 180,E1 -8234.528,E2 -8234.528} C_VEL
LIN {X 0,Y 453.439,Z 146.998,A -85,B 0,C 180,E1 -8238.071,E2 -8238.071} C_VEL
LIN {X 0,Y 453.468,Z 146.998,A -85,B 0,C 180,E1 -8240.798,E2 -8240.798} C_VEL
LIN {X 0,Y 453.454,Z 146.997,A -85,B 0,C 180,E1 -8243.917,E2 -8243.917} C_VEL
LIN {X 0,Y 453.476,Z 146.999,A -85,B 0,C 180,E1 -8247.15,E2 -8247.15} C_VEL
LIN {X 0,Y 453.46,Z 146.997,A -85,B 0,C 180,E1 -8250.267,E2 -8250.267} C_VEL
LIN {X 0,Y 453.458,Z 146.998,A -85,B 0,C 180,E1 -8253.291,E2 -8253.291} C_VEL
LIN {X 0,Y 453.495,Z 146.993,A -85,B 0,C 180,E1 -8256.238,E2 -8256.238} C_VEL
LIN {X 0,Y 453.478,Z 146.996,A -85,B 0,C 180,E1 -8259.117,E2 -8259.117} C_VEL
LIN {X 0,Y 453.487,Z 146.993,A -85,B 0,C 180,E1 -8261.943,E2 -8261.943} C_VEL
LIN {X 0,Y 453.52,Z 146.994,A -85,B 0,C 180,E1 -8264.726,E2 -8264.726} C_VEL
LIN {X 0,Y 453.562,Z 146.99,A -85,B 0,C 180,E1 -8268.379,E2 -8268.379} C_VEL
LIN {X 0,Y 453.569,Z 146.983,A -85,B 0,C 180,E1 -8271.086,E2 -8271.086} C_VEL
LIN {X 0,Y 453.639,Z 146.975,A -85,B 0,C 180,E1 -8273.774,E2 -8273.774} C_VEL
LIN {X 0,Y 453.707,Z 146.965,A -85,B 0,C 180,E1 -8277.336,E2 -8277.336} C_VEL
LIN {X 0,Y 453.771,Z 146.962,A -85,B 0,C 180,E1 -8280,E2 -8280} C_VEL
LIN {X 0,Y 453.706,Z 146.967,A -85,B 0,C 180,E1 -8282.664,E2 -8282.664} C_VEL
LIN {X 0,Y 453.638,Z 146.979,A -85,B 0,C 180,E1 -8286.226,E2 -8286.226} C_VEL
LIN {X 0,Y 453.562,Z 146.983,A -85,B 0,C 180,E1 -8288.914,E2 -8288.914} C_VEL
LIN {X 0,Y 453.568,Z 146.983,A -85,B 0,C 180,E1 -8292.529,E2 -8292.529} C_VEL
LIN {X 0,Y 453.489,Z 146.995,A -85,B 0,C 180,E1 -8296.198,E2 -8296.198} C_VEL
LIN {X 0,Y 453.489,Z 146.993,A -85,B 0,C 180,E1 -8299.027,E2 -8299.027} C_VEL
LIN {X 0,Y 453.47,Z 147,A -85,B 0,C 180,E1 -8301.836,E2 -8301.836} C_VEL
LIN {X 0,Y 453.464,Z 146.995,A -85,B 0,C 180,E1 -8304.737,E2 -8304.737} C_VEL
LIN {X 0,Y 453.458,Z 146.998,A -85,B 0,C 180,E1 -8307.941,E2 -8307.941} C_VEL
LIN {X 0,Y 453.449,Z 146.998,A -85,B 0,C 180,E1 -8310.762,E2 -8310.762} C_VEL
LIN {X 0,Y 453.457,Z 146.998,A -85,B 0,C 180,E1 -8313.915,E2 -8313.915} C_VEL
LIN {X 0,Y 453.436,Z 147.005,A -85,B 0,C 180,E1 -8317.191,E2 -8317.191} C_VEL
LIN {X 0,Y 453.471,Z 146.996,A -85,B 0,C 180,E1 -8320.612,E2 -8320.612} C_VEL
LIN {X 0,Y 453.482,Z 146.994,A -85,B 0,C 180,E1 -8324.528,E2 -8324.528} C_VEL
LIN {X 0,Y 453.435,Z 146.999,A -85,B 0,C 180,E1 -8328.071,E2 -8328.071} C_VEL
LIN {X 0,Y 453.431,Z 147.005,A -85,B 0,C 180,E1 -8330.803,E2 -8330.803} C_VEL
LIN {X 0,Y 453.44,Z 146.998,A -85,B 0,C 180,E1 -8333.915,E2 -8333.915} C_VEL
LIN {X 0,Y 453.466,Z 147.003,A -85,B 0,C 180,E1 -8336.816,E2 -8336.816} C_VEL
LIN {X 0,Y 453.448,Z 147.003,A -85,B 0,C 180,E1 -8340.266,E2 -8340.266} C_VEL
LIN {X 0,Y 453.424,Z 147.007,A -85,B 0,C 180,E1 -8343.288,E2 -8343.288} C_VEL
LIN {X 0,Y 453.479,Z 147.118,A -85,B 0,C 180,E1 -8343.978,E2 -8343.978} C_VEL
LIN {X 0,Y 455.722,Z 158.938,A -85,B 0,C 180,E1 -8346.361,E2 -8346.361} C_VEL
LIN {X 0,Y 455.559,Z 167.092,A -85,B 0,C 180,E1 -8347.892,E2 -8347.892} C_VEL
LIN {X 0,Y 454.725,Z 184.292,A -85,B 0,C 180,E1 -8351.061,E2 -8351.061} C_VEL
LIN {X 0,Y 454.369,Z 192.065,A -85,B 0,C 180,E1 -8352.479,E2 -8352.479} C_VEL
LIN {X 0,Y 457.488,Z 212.293,A -85,B 0,C 180,E1 -8352.937,E2 -8352.937} C_VEL
LIN {X 0,Y 456.713,Z 300.615,A -85,B 0,C 180,E1 -8354.378,E2 -8354.378} C_VEL
LIN {X 0,Y 456.304,Z 314.464,A -85,B 0,C 180,E1 -8354.792,E2 -8354.792} C_VEL
LIN {X 0,Y 455.803,Z 327.416,A -85,B 0,C 180,E1 -8355.375,E2 -8355.375} C_VEL
LIN {X 0,Y 455.2,Z 339.997,A -85,B 0,C 180,E1 -8356.154,E2 -8356.154} C_VEL
LIN {X 0,Y 454.647,Z 351.04,A -85,B 0,C 180,E1 -8357.031,E2 -8357.031} C_VEL
LIN {X 0,Y 454.208,Z 360.312,A -85,B 0,C 180,E1 -8357.943,E2 -8357.943} C_VEL
LIN {X 0,Y 453.654,Z 369.632,A -85,B 0,C 180,E1 -8359.06,E2 -8359.06} C_VEL
LIN {X 0,Y 453.207,Z 378.672,A -85,B 0,C 180,E1 -8360.404,E2 -8360.404} C_VEL
LIN {X 0,Y 452.902,Z 385.954,A -85,B 0,C 180,E1 -8361.747,E2 -8361.747} C_VEL
LIN {X 0,Y 452.681,Z 390.87,A -85,B 0,C 180,E1 -8362.865,E2 -8362.865} C_VEL
LIN {X 0,Y 452.552,Z 395.644,A -85,B 0,C 180,E1 -8364.206,E2 -8364.206} C_VEL
LIN {X 0,Y 452.485,Z 399.294,A -85,B 0,C 180,E1 -8365.546,E2 -8365.546} C_VEL
LIN {X 0,Y 452.479,Z 401.178,A -85,B 0,C 180,E1 -8366.438,E2 -8366.438} C_VEL
LIN {X 0,Y 452.508,Z 402.595,A -85,B 0,C 180,E1 -8367.329,E2 -8367.329} C_VEL
LIN {X 0,Y 452.429,Z 404.212,A -85,B 0,C 180,E1 -8369.11,E2 -8369.11} C_VEL
LIN {X 0,Y 452.437,Z 404.435,A -85,B 0,C 180,E1 -8370,E2 -8370} C_VEL
LIN {X 0,Y 452.429,Z 404.222,A -85,B 0,C 180,E1 -8370.89,E2 -8370.89} C_VEL
LIN {X 0,Y 452.508,Z 402.611,A -85,B 0,C 180,E1 -8372.671,E2 -8372.671} C_VEL
LIN {X 0,Y 452.479,Z 401.208,A -85,B 0,C 180,E1 -8373.562,E2 -8373.562} C_VEL
LIN {X 0,Y 452.543,Z 398.256,A -85,B 0,C 180,E1 -8374.9,E2 -8374.9} C_VEL
LIN {X 0,Y 452.611,Z 393.723,A -85,B 0,C 180,E1 -8376.396,E2 -8376.396} C_VEL
LIN {X 0,Y 452.808,Z 388.12,A -85,B 0,C 180,E1 -8377.805,E2 -8377.805} C_VEL
LIN {X 0,Y 453.085,Z 381.409,A -85,B 0,C 180,E1 -8379.149,E2 -8379.149} C_VEL
LIN {X 0,Y 453.468,Z 373.089,A -85,B 0,C 180,E1 -8380.493,E2 -8380.493} C_VEL
LIN {X 0,Y 454.03,Z 364.565,A -85,B 0,C 180,E1 -8381.609,E2 -8381.609} C_VEL
LIN {X 0,Y 454.535,Z 354.903,A -85,B 0,C 180,E1 -8382.645,E2 -8382.645} C_VEL
LIN {X 0,Y 455.092,Z 343.62,A -85,B 0,C 180,E1 -8383.622,E2 -8383.622} C_VEL
LIN {X 0,Y 455.626,Z 332.207,A -85,B 0,C 180,E1 -8384.402,E2 -8384.402} C_VEL
LIN {X 0,Y 456.187,Z 320.475,A -85,B 0,C 180,E1 -8385.012,E2 -8385.012} C_VEL
LIN {X 0,Y 456.658,Z 306.995,A -85,B 0,C 180,E1 -8385.51,E2 -8385.51} C_VEL
LIN {X 0,Y 457.016,Z 293.625,A -85,B 0,C 180,E1 -8385.812,E2 -8385.812} C_VEL
LIN {X 0,Y 457.567,Z 211.427,A -85,B 0,C 180,E1 -8387.146,E2 -8387.146} C_VEL
LIN {X 0,Y 454.41,Z 191.524,A -85,B 0,C 180,E1 -8387.626,E2 -8387.626} C_VEL
LIN {X 0,Y 455.097,Z 175.338,A -85,B 0,C 180,E1 -8390.569,E2 -8390.569} C_VEL
LIN {X 0,Y 455.851,Z 160.013,A -85,B 0,C 180,E1 -8393.391,E2 -8393.391} C_VEL
LIN {X 0,Y 454.055,Z 149.733,A -85,B 0,C 180,E1 -8395.438,E2 -8395.438} C_VEL
LIN {X 0,Y 453.472,Z 146.999,A -85,B 0,C 180,E1 -8396.045,E2 -8396.045} C_VEL
LIN {X 0,Y 453.449,Z 147.004,A -85,B 0,C 180,E1 -8398.716,E2 -8398.716} C_VEL
LIN {X 0,Y 453.436,Z 147.006,A -85,B 0,C 180,E1 -8401.802,E2 -8401.802} C_VEL
LIN {X 0,Y 453.468,Z 147.002,A -85,B 0,C 180,E1 -8404.991,E2 -8404.991} C_VEL
LIN {X 0,Y 453.439,Z 147,A -85,B 0,C 180,E1 -8408.315,E2 -8408.315} C_VEL
LIN {X 0,Y 453.465,Z 146.999,A -85,B 0,C 180,E1 -8410.613,E2 -8410.613} C_VEL
LIN {X 0,Y 453.482,Z 146.997,A -85,B 0,C 180,E1 -8414.528,E2 -8414.528} C_VEL
LIN {X 0,Y 453.432,Z 147,A -85,B 0,C 180,E1 -8418.072,E2 -8418.072} C_VEL
LIN {X 0,Y 453.425,Z 147.004,A -85,B 0,C 180,E1 -8420.805,E2 -8420.805} C_VEL
LIN {X 0,Y 453.44,Z 146.997,A -85,B 0,C 180,E1 -8423.916,E2 -8423.916} C_VEL
LIN {X 0,Y 453.467,Z 146.997,A -85,B 0,C 180,E1 -8426.816,E2 -8426.816} C_VEL
LIN {X 0,Y 453.45,Z 146.999,A -85,B 0,C 180,E1 -8430.266,E2 -8430.266} C_VEL
LIN {X 0,Y 453.426,Z 147.001,A -85,B 0,C 180,E1 -8433.289,E2 -8433.289} C_VEL
LIN {X 0,Y 453.473,Z 146.994,A -85,B 0,C 180,E1 -8436.237,E2 -8436.237} C_VEL
LIN {X 0,Y 453.44,Z 146.994,A -85,B 0,C 180,E1 -8439.116,E2 -8439.116} C_VEL
LIN {X 0,Y 453.459,Z 146.998,A -85,B 0,C 180,E1 -8441.942,E2 -8441.942} C_VEL
LIN {X 0,Y 453.488,Z 146.995,A -85,B 0,C 180,E1 -8444.725,E2 -8444.725} C_VEL
LIN {X 0,Y 453.569,Z 146.982,A -85,B 0,C 180,E1 -8447.471,E2 -8447.471} C_VEL
LIN {X 0,Y 453.559,Z 146.984,A -85,B 0,C 180,E1 -8451.086,E2 -8451.086} C_VEL
LIN {X 0,Y 453.632,Z 146.971,A -85,B 0,C 180,E1 -8453.774,E2 -8453.774} C_VEL
LIN {X 0,Y 453.705,Z 146.962,A -85,B 0,C 180,E1 -8457.336,E2 -8457.336} C_VEL
LIN {X 0,Y 453.771,Z 146.962,A -85,B 0,C 180,E1 -8460,E2 -8460} C_VEL
LIN {X 0,Y 453.705,Z 146.966,A -85,B 0,C 180,E1 -8462.664,E2 -8462.664} C_VEL
LIN {X 0,Y 453.639,Z 146.977,A -85,B 0,C 180,E1 -8466.226,E2 -8466.226} C_VEL
LIN {X 0,Y 453.562,Z 146.982,A -85,B 0,C 180,E1 -8468.914,E2 -8468.914} C_VEL
LIN {X 0,Y 453.569,Z 146.982,A -85,B 0,C 180,E1 -8472.529,E2 -8472.529} C_VEL
LIN {X 0,Y 453.5,Z 146.996,A -85,B 0,C 180,E1 -8476.198,E2 -8476.198} C_VEL
LIN {X 0,Y 453.489,Z 146.994,A -85,B 0,C 180,E1 -8479.027,E2 -8479.027} C_VEL
LIN {X 0,Y 453.475,Z 147.001,A -85,B 0,C 180,E1 -8481.836,E2 -8481.836} C_VEL
LIN {X 0,Y 453.473,Z 146.997,A -85,B 0,C 180,E1 -8484.737,E2 -8484.737} C_VEL
LIN {X 0,Y 453.464,Z 147.003,A -85,B 0,C 180,E1 -8487.942,E2 -8487.942} C_VEL
LIN {X 0,Y 453.458,Z 147,A -85,B 0,C 180,E1 -8490.761,E2 -8490.761} C_VEL
LIN {X 0,Y 453.47,Z 147.003,A -85,B 0,C 180,E1 -8493.913,E2 -8493.913} C_VEL
LIN {X 0,Y 453.494,Z 147.014,A -85,B 0,C 180,E1 -8495.874,E2 -8495.874} C_VEL
LIN {X 0,Y 454.943,Z 154.696,A -85,B 0,C 180,E1 -8497.548,E2 -8497.548} C_VEL
LIN {X 0,Y 454.947,Z 161.804,A -85,B 0,C 180,E1 -8499.014,E2 -8499.014} C_VEL
LIN {X 0,Y 454.683,Z 168.859,A -85,B 0,C 180,E1 -8500.445,E2 -8500.445} C_VEL
LIN {X 0,Y 457.9,Z 185.54,A -85,B 0,C 180,E1 -8500.873,E2 -8500.873} C_VEL
LIN {X 0,Y 456.93,Z 276.891,A -85,B 0,C 180,E1 -8502.373,E2 -8502.373} C_VEL
LIN {X 0,Y 456.653,Z 290.3,A -85,B 0,C 180,E1 -8502.783,E2 -8502.783} C_VEL
LIN {X 0,Y 456.218,Z 303.246,A -85,B 0,C 180,E1 -8503.371,E2 -8503.371} C_VEL
LIN {X 0,Y 455.66,Z 315.005,A -85,B 0,C 180,E1 -8504.096,E2 -8504.096} C_VEL
LIN {X 0,Y 455.098,Z 327.063,A -85,B 0,C 180,E1 -8505.057,E2 -8505.057} C_VEL
LIN {X 0,Y 454.501,Z 337.531,A -85,B 0,C 180,E1 -8506.117,E2 -8506.117} C_VEL
LIN {X 0,Y 453.979,Z 347.217,A -85,B 0,C 180,E1 -8507.337,E2 -8507.337} C_VEL
LIN {X 0,Y 453.547,Z 354.832,A -85,B 0,C 180,E1 -8508.513,E2 -8508.513} C_VEL
LIN {X 0,Y 453.127,Z 362.421,A -85,B 0,C 180,E1 -8509.971,E2 -8509.971} C_VEL
LIN {X 0,Y 452.881,Z 367.728,A -85,B 0,C 180,E1 -8511.252,E2 -8511.252} C_VEL
LIN {X 0,Y 452.657,Z 372.503,A -85,B 0,C 180,E1 -8512.733,E2 -8512.733} C_VEL
LIN {X 0,Y 452.554,Z 375.276,A -85,B 0,C 180,E1 -8513.857,E2 -8513.857} C_VEL
LIN {X 0,Y 452.383,Z 377.951,A -85,B 0,C 180,E1 -8515.425,E2 -8515.425} C_VEL
LIN {X 0,Y 452.333,Z 379.397,A -85,B 0,C 180,E1 -8517.057,E2 -8517.057} C_VEL
LIN {X 0,Y 452.333,Z 379.52,A -85,B 0,C 180,E1 -8518.71,E2 -8518.71} C_VEL
LIN {X 0,Y 452.431,Z 378.125,A -85,B 0,C 180,E1 -8520.447,E2 -8520.447} C_VEL
LIN {X 0,Y 452.534,Z 375.123,A -85,B 0,C 180,E1 -8522.231,E2 -8522.231} C_VEL
LIN {X 0,Y 452.723,Z 371.179,A -85,B 0,C 180,E1 -8523.741,E2 -8523.741} C_VEL
LIN {X 0,Y 452.893,Z 367.903,A -85,B 0,C 180,E1 -8524.712,E2 -8524.712} C_VEL
LIN {X 0,Y 452.365,Z 365.395,A -85,B 0,C 180,E1 -8525.386,E2 -8525.386} C_VEL
LIN {X 0,Y 449.75,Z 360.898,A -85,B 0,C 180,E1 -8526.458,E2 -8526.458} C_VEL
LIN {X 0,Y 447.131,Z 355.763,A -85,B 0,C 180,E1 -8527.493,E2 -8527.493} C_VEL
LIN {X 0,Y 446.607,Z 352.25,A -85,B 0,C 180,E1 -8528.102,E2 -8528.102} C_VEL
LIN {X 0,Y 447.075,Z 344.12,A -85,B 0,C 180,E1 -8529.286,E2 -8529.286} C_VEL
LIN {X 0,Y 447.649,Z 334.833,A -85,B 0,C 180,E1 -8530.389,E2 -8530.389} C_VEL
LIN {X 0,Y 448.121,Z 324.796,A -85,B 0,C 180,E1 -8531.364,E2 -8531.364} C_VEL
LIN {X 0,Y 448.721,Z 313.861,A -85,B 0,C 180,E1 -8532.217,E2 -8532.217} C_VEL
LIN {X 0,Y 449.198,Z 301.959,A -85,B 0,C 180,E1 -8532.941,E2 -8532.941} C_VEL
LIN {X 0,Y 449.634,Z 289.076,A -85,B 0,C 180,E1 -8533.513,E2 -8533.513} C_VEL
LIN {X 0,Y 449.991,Z 275.859,A -85,B 0,C 180,E1 -8533.905,E2 -8533.905} C_VEL
LIN {X 0,Y 450.796,Z 185.502,A -85,B 0,C 180,E1 -8535.401,E2 -8535.401} C_VEL
LIN {X 0,Y 447.639,Z 168.905,A -85,B 0,C 180,E1 -8535.817,E2 -8535.817} C_VEL
LIN {X 0,Y 448.049,Z 156.501,A -85,B 0,C 180,E1 -8538.463,E2 -8538.463} C_VEL
LIN {X 0,Y 446.551,Z 147.863,A -85,B 0,C 180,E1 -8540.431,E2 -8540.431} C_VEL
LIN {X 0,Y 446.612,Z 147.853,A -85,B 0,C 180,E1 -8543.676,E2 -8543.676} C_VEL
LIN {X 0,Y 446.683,Z 147.84,A -85,B 0,C 180,E1 -8547.295,E2 -8547.295} C_VEL
LIN {X 0,Y 446.764,Z 147.833,A -85,B 0,C 180,E1 -8550,E2 -8550} C_VEL
LIN {X 0,Y 446.657,Z 147.846,A -85,B 0,C 180,E1 -8552.706,E2 -8552.706} C_VEL
LIN {X 0,Y 446.609,Z 147.856,A -85,B 0,C 180,E1 -8556.324,E2 -8556.324} C_VEL
LIN {X 0,Y 446.529,Z 147.859,A -85,B 0,C 180,E1 -8559.056,E2 -8559.056} C_VEL
LIN {X 0,Y 446.524,Z 147.861,A -85,B 0,C 180,E1 -8562.73,E2 -8562.73} C_VEL
LIN {X 0,Y 446.456,Z 147.873,A -85,B 0,C 180,E1 -8566.209,E2 -8566.209} C_VEL
LIN {X 0,Y 446.471,Z 147.868,A -85,B 0,C 180,E1 -8569.303,E2 -8569.303} C_VEL
LIN {X 0,Y 446.42,Z 147.876,A -85,B 0,C 180,E1 -8572.2,E2 -8572.2} C_VEL
LIN {X 0,Y 446.424,Z 147.873,A -85,B 0,C 180,E1 -8575.155,E2 -8575.155} C_VEL
LIN {X 0,Y 446.439,Z 147.872,A -85,B 0,C 180,E1 -8578.182,E2 -8578.182} C_VEL
LIN {X 0,Y 446.417,Z 147.877,A -85,B 0,C 180,E1 -8581.301,E2 -8581.301} C_VEL
LIN {X 0,Y 446.424,Z 147.872,A -85,B 0,C 180,E1 -8584.524,E2 -8584.524} C_VEL
LIN {X 0,Y 446.413,Z 147.875,A -85,B 0,C 180,E1 -8588.078,E2 -8588.078} C_VEL
LIN {X 0,Y 446.403,Z 147.883,A -85,B 0,C 180,E1 -8591.394,E2 -8591.394} C_VEL
LIN {X 0,Y 446.452,Z 147.874,A -85,B 0,C 180,E1 -8595.104,E2 -8595.104} C_VEL
LIN {X 0,Y 446.403,Z 147.876,A -85,B 0,C 180,E1 -8598.606,E2 -8598.606} C_VEL
LIN {X 0,Y 446.413,Z 147.874,A -85,B 0,C 180,E1 -8601.922,E2 -8601.922} C_VEL
LIN {X 0,Y 446.425,Z 147.874,A -85,B 0,C 180,E1 -8605.476,E2 -8605.476} C_VEL
LIN {X 0,Y 446.41,Z 147.878,A -85,B 0,C 180,E1 -8608.699,E2 -8608.699} C_VEL
LIN {X 0,Y 446.429,Z 147.872,A -85,B 0,C 180,E1 -8611.836,E2 -8611.836} C_VEL
LIN {X 0,Y 446.425,Z 147.879,A -85,B 0,C 180,E1 -8614.846,E2 -8614.846} C_VEL
LIN {X 0,Y 446.45,Z 147.871,A -85,B 0,C 180,E1 -8618.246,E2 -8618.246} C_VEL
LIN {X 0,Y 446.442,Z 147.87,A -85,B 0,C 180,E1 -8621.648,E2 -8621.648} C_VEL
LIN {X 0,Y 446.462,Z 147.874,A -85,B 0,C 180,E1 -8624.478,E2 -8624.478} C_VEL
LIN {X 0,Y 446.521,Z 147.86,A -85,B 0,C 180,E1 -8627.384,E2 -8627.384} C_VEL
LIN {X 0,Y 446.52,Z 147.862,A -85,B 0,C 180,E1 -8630.944,E2 -8630.944} C_VEL
LIN {X 0,Y 446.609,Z 147.85,A -85,B 0,C 180,E1 -8633.676,E2 -8633.676} C_VEL
LIN {X 0,Y 446.656,Z 147.843,A -85,B 0,C 180,E1 -8637.294,E2 -8637.294} C_VEL
LIN {X 0,Y 446.722,Z 147.84,A -85,B 0,C 180,E1 -8640,E2 -8640} C_VEL
LIN {X 0,Y 446.655,Z 147.845,A -85,B 0,C 180,E1 -8642.706,E2 -8642.706} C_VEL
LIN {X 0,Y 446.609,Z 147.853,A -85,B 0,C 180,E1 -8646.324,E2 -8646.324} C_VEL
LIN {X 0,Y 446.512,Z 147.861,A -85,B 0,C 180,E1 -8649.056,E2 -8649.056} C_VEL
LIN {X 0,Y 446.496,Z 147.863,A -85,B 0,C 180,E1 -8652.73,E2 -8652.73} C_VEL
LIN {X 0,Y 446.458,Z 147.871,A -85,B 0,C 180,E1 -8656.209,E2 -8656.209} C_VEL
LIN {X 0,Y 446.43,Z 147.874,A -85,B 0,C 180,E1 -8659.305,E2 -8659.305} C_VEL
LIN {X 0,Y 446.408,Z 147.876,A -85,B 0,C 180,E1 -8662.2,E2 -8662.2} C_VEL
LIN {X 0,Y 446.415,Z 147.876,A -85,B 0,C 180,E1 -8665.155,E2 -8665.155} C_VEL
LIN {X 0,Y 446.418,Z 147.874,A -85,B 0,C 180,E1 -8668.183,E2 -8668.183} C_VEL
LIN {X 0,Y 446.391,Z 147.882,A -85,B 0,C 180,E1 -8671.302,E2 -8671.302} C_VEL
LIN {X 0,Y 446.415,Z 147.873,A -85,B 0,C 180,E1 -8674.524,E2 -8674.524} C_VEL
LIN {X 0,Y 446.397,Z 147.876,A -85,B 0,C 180,E1 -8678.076,E2 -8678.076} C_VEL
LIN {X 0,Y 446.401,Z 147.88,A -85,B 0,C 180,E1 -8681.394,E2 -8681.394} C_VEL
LIN {X 0,Y 446.451,Z 147.877,A -85,B 0,C 180,E1 -8685.104,E2 -8685.104} C_VEL
LIN {X 0,Y 446.399,Z 147.878,A -85,B 0,C 180,E1 -8688.605,E2 -8688.605} C_VEL
LIN {X 0,Y 446.396,Z 147.876,A -85,B 0,C 180,E1 -8691.924,E2 -8691.924} C_VEL
LIN {X 0,Y 446.413,Z 147.875,A -85,B 0,C 180,E1 -8695.475,E2 -8695.475} C_VEL
LIN {X 0,Y 446.39,Z 147.884,A -85,B 0,C 180,E1 -8698.697,E2 -8698.697} C_VEL
LIN {X 0,Y 446.402,Z 147.878,A -85,B 0,C 180,E1 -8701.842,E2 -8701.842} C_VEL
LIN {X 0,Y 446.423,Z 148.03,A -85,B 0,C 180,E1 -8703.766,E2 -8703.766} C_VEL
LIN {X 0,Y 448.538,Z 158.682,A -85,B 0,C 180,E1 -8705.959,E2 -8705.959} C_VEL
LIN {X 0,Y 448.887,Z 162.509,A -85,B 0,C 180,E1 -8706.713,E2 -8706.713} C_VEL
LIN {X 0,Y 447.939,Z 181.518,A -85,B 0,C 180,E1 -8710.285,E2 -8710.285} C_VEL
LIN {X 0,Y 447.416,Z 191.896,A -85,B 0,C 180,E1 -8712.21,E2 -8712.21} C_VEL
LIN {X 0,Y 450.681,Z 213.502,A -85,B 0,C 180,E1 -8712.706,E2 -8712.706} C_VEL
LIN {X 0,Y 449.877,Z 299.924,A -85,B 0,C 180,E1 -8714.134,E2 -8714.134} C_VEL
LIN {X 0,Y 449.49,Z 313.176,A -85,B 0,C 180,E1 -8714.527,E2 -8714.527} C_VEL
LIN {X 0,Y 448.936,Z 325.913,A -85,B 0,C 180,E1 -8715.088,E2 -8715.088} C_VEL
LIN {X 0,Y 448.363,Z 338.048,A -85,B 0,C 180,E1 -8715.823,E2 -8715.823} C_VEL
LIN {X 0,Y 447.778,Z 349.071,A -85,B 0,C 180,E1 -8716.683,E2 -8716.683} C_VEL
LIN {X 0,Y 447.224,Z 360.011,A -85,B 0,C 180,E1 -8717.752,E2 -8717.752} C_VEL
LIN {X 0,Y 446.665,Z 369.361,A -85,B 0,C 180,E1 -8718.887,E2 -8718.887} C_VEL
LIN {X 0,Y 446.178,Z 378.418,A -85,B 0,C 180,E1 -8720.251,E2 -8720.251} C_VEL
LIN {X 0,Y 445.84,Z 385.713,A -85,B 0,C 180,E1 -8721.616,E2 -8721.616} C_VEL
LIN {X 0,Y 445.612,Z 390.64,A -85,B 0,C 180,E1 -8722.751,E2 -8722.751} C_VEL
LIN {X 0,Y 445.467,Z 394.93,A -85,B 0,C 180,E1 -8723.958,E2 -8723.958} C_VEL
LIN {X 0,Y 445.41,Z 399.081,A -85,B 0,C 180,E1 -8725.475,E2 -8725.475} C_VEL
LIN {X 0,Y 445.378,Z 400.969,A -85,B 0,C 180,E1 -8726.381,E2 -8726.381} C_VEL
LIN {X 0,Y 445.433,Z 402.392,A -85,B 0,C 180,E1 -8727.287,E2 -8727.287} C_VEL
LIN {X 0,Y 445.34,Z 404.014,A -85,B 0,C 180,E1 -8729.096,E2 -8729.096} C_VEL
LIN {X 0,Y 445.344,Z 404.24,A -85,B 0,C 180,E1 -8730,E2 -8730} C_VEL
LIN {X 0,Y 445.34,Z 404.031,A -85,B 0,C 180,E1 -8730.904,E2 -8730.904} C_VEL
LIN {X 0,Y 445.433,Z 402.423,A -85,B 0,C 180,E1 -8732.713,E2 -8732.713} C_VEL
LIN {X 0,Y 445.377,Z 401.021,A -85,B 0,C 180,E1 -8733.619,E2 -8733.619} C_VEL
LIN {X 0,Y 445.471,Z 398.072,A -85,B 0,C 180,E1 -8734.978,E2 -8734.978} C_VEL
LIN {X 0,Y 445.53,Z 393.933,A -85,B 0,C 180,E1 -8736.386,E2 -8736.386} C_VEL
LIN {X 0,Y 445.733,Z 387.947,A -85,B 0,C 180,E1 -8737.93,E2 -8737.93} C_VEL
LIN {X 0,Y 446.058,Z 381.244,A -85,B 0,C 180,E1 -8739.294,E2 -8739.294} C_VEL
LIN {X 0,Y 446.465,Z 372.929,A -85,B 0,C 180,E1 -8740.659,E2 -8740.659} C_VEL
LIN {X 0,Y 447.04,Z 364.413,A -85,B 0,C 180,E1 -8741.793,E2 -8741.793} C_VEL
LIN {X 0,Y 447.667,Z 353.686,A -85,B 0,C 180,E1 -8742.947,E2 -8742.947} C_VEL
LIN {X 0,Y 448.263,Z 342.063,A -85,B 0,C 180,E1 -8743.949,E2 -8743.949} C_VEL
LIN {X 0,Y 448.852,Z 330.176,A -85,B 0,C 180,E1 -8744.74,E2 -8744.74} C_VEL
LIN {X 0,Y 449.47,Z 317.836,A -85,B 0,C 180,E1 -8745.357,E2 -8745.357} C_VEL
LIN {X 0,Y 449.9,Z 305.21,A -85,B 0,C 180,E1 -8745.807,E2 -8745.807} C_VEL
LIN {X 0,Y 450.214,Z 290.409,A -85,B 0,C 180,E1 -8746.115,E2 -8746.115} C_VEL
LIN {X 0,Y 450.846,Z 212.586,A -85,B 0,C 180,E1 -8747.398,E2 -8747.398} C_VEL
LIN {X 0,Y 447.466,Z 191.32,A -85,B 0,C 180,E1 -8747.92,E2 -8747.92} C_VEL
LIN {X 0,Y 448.286,Z 173.931,A -85,B 0,C 180,E1 -8751.136,E2 -8751.136} C_VEL
LIN {X 0,Y 448.921,Z 161.154,A -85,B 0,C 180,E1 -8753.529,E2 -8753.529} C_VEL
LIN {X 0,Y 446.797,Z 149.611,A -85,B 0,C 180,E1 -8755.881,E2 -8755.881} C_VEL
LIN {X 0,Y 446.389,Z 147.881,A -85,B 0,C 180,E1 -8756.27,E2 -8756.27} C_VEL
LIN {X 0,Y 446.409,Z 147.883,A -85,B 0,C 180,E1 -8759.213,E2 -8759.213} C_VEL
LIN {X 0,Y 446.398,Z 147.882,A -85,B 0,C 180,E1 -8762.364,E2 -8762.364} C_VEL
LIN {X 0,Y 446.407,Z 147.879,A -85,B 0,C 180,E1 -8765.628,E2 -8765.628} C_VEL
LIN {X 0,Y 446.387,Z 147.885,A -85,B 0,C 180,E1 -8769.033,E2 -8769.033} C_VEL
LIN {X 0,Y 446.378,Z 147.88,A -85,B 0,C 180,E1 -8772.269,E2 -8772.269} C_VEL
LIN {X 0,Y 446.451,Z 147.877,A -85,B 0,C 180,E1 -8775.104,E2 -8775.104} C_VEL
LIN {X 0,Y 446.397,Z 147.88,A -85,B 0,C 180,E1 -8778.605,E2 -8778.605} C_VEL
LIN {X 0,Y 446.388,Z 147.878,A -85,B 0,C 180,E1 -8782.119,E2 -8782.119} C_VEL
LIN {X 0,Y 446.414,Z 147.875,A -85,B 0,C 180,E1 -8785.476,E2 -8785.476} C_VEL
LIN {X 0,Y 446.391,Z 147.882,A -85,B 0,C 180,E1 -8788.698,E2 -8788.698} C_VEL
LIN {X 0,Y 446.403,Z 147.873,A -85,B 0,C 180,E1 -8791.842,E2 -8791.842} C_VEL
LIN {X 0,Y 446.409,Z 147.874,A -85,B 0,C 180,E1 -8794.845,E2 -8794.845} C_VEL
LIN {X 0,Y 446.445,Z 147.874,A -85,B 0,C 180,E1 -8798.248,E2 -8798.248} C_VEL
LIN {X 0,Y 446.413,Z 147.875,A -85,B 0,C 180,E1 -8801.647,E2 -8801.647} C_VEL
LIN {X 0,Y 446.431,Z 147.872,A -85,B 0,C 180,E1 -8804.477,E2 -8804.477} C_VEL
LIN {X 0,Y 446.52,Z 147.86,A -85,B 0,C 180,E1 -8807.384,E2 -8807.384} C_VEL
LIN {X 0,Y 446.51,Z 147.862,A -85,B 0,C 180,E1 -8810.944,E2 -8810.944} C_VEL
LIN {X 0,Y 446.603,Z 147.845,A -85,B 0,C 180,E1 -8813.676,E2 -8813.676} C_VEL
LIN {X 0,Y 446.655,Z 147.84,A -85,B 0,C 180,E1 -8817.294,E2 -8817.294} C_VEL
LIN {X 0,Y 446.722,Z 147.84,A -85,B 0,C 180,E1 -8820,E2 -8820} C_VEL
LIN {X 0,Y 446.655,Z 147.844,A -85,B 0,C 180,E1 -8822.706,E2 -8822.706} C_VEL
LIN {X 0,Y 446.609,Z 147.854,A -85,B 0,C 180,E1 -8826.324,E2 -8826.324} C_VEL
LIN {X 0,Y 446.513,Z 147.86,A -85,B 0,C 180,E1 -8829.056,E2 -8829.056} C_VEL
LIN {X 0,Y 446.526,Z 147.859,A -85,B 0,C 180,E1 -8832.73,E2 -8832.73} C_VEL
LIN {X 0,Y 446.454,Z 147.874,A -85,B 0,C 180,E1 -8836.207,E2 -8836.207} C_VEL
LIN {X 0,Y 446.435,Z 147.874,A -85,B 0,C 180,E1 -8839.305,E2 -8839.305} C_VEL
LIN {X 0,Y 446.416,Z 147.877,A -85,B 0,C 180,E1 -8842.2,E2 -8842.2} C_VEL
LIN {X 0,Y 446.425,Z 147.877,A -85,B 0,C 180,E1 -8845.154,E2 -8845.154} C_VEL
LIN {X 0,Y 446.42,Z 147.878,A -85,B 0,C 180,E1 -8848.183,E2 -8848.183} C_VEL
LIN {X 0,Y 446.411,Z 147.88,A -85,B 0,C 180,E1 -8851.301,E2 -8851.301} C_VEL
LIN {X 0,Y 446.426,Z 147.878,A -85,B 0,C 180,E1 -8854.524,E2 -8854.524} C_VEL
LIN {X 0,Y 446.457,Z 147.947,A -85,B 0,C 180,E1 -8855.657,E2 -8855.657} C_VEL
LIN {X 0,Y 448.127,Z 157.223,A -85,B 0,C 180,E1 -8857.708,E2 -8857.708} C_VEL
LIN {X 0,Y 447.813,Z 169.117,A -85,B 0,C 180,E1 -8860.16,E2 -8860.16} C_VEL
LIN {X 0,Y 451.183,Z 187.14,A -85,B 0,C 180,E1 -8860.622,E2 -8860.622} C_VEL
LIN {X 0,Y 450.148,Z 276.554,A -85,B 0,C 180,E1 -8862.109,E2 -8862.109} C_VEL
LIN {X 0,Y 449.829,Z 289.972,A -85,B 0,C 180,E1 -8862.518,E2 -8862.518} C_VEL
LIN {X 0,Y 449.444,Z 302.065,A -85,B 0,C 180,E1 -8863.062,E2 -8863.062} C_VEL
LIN {X 0,Y 448.834,Z 314.41,A -85,B 0,C 180,E1 -8863.814,E2 -8863.814} C_VEL
LIN {X 0,Y 448.255,Z 325.641,A -85,B 0,C 180,E1 -8864.703,E2 -8864.703} C_VEL
LIN {X 0,Y 447.697,Z 335.636,A -85,B 0,C 180,E1 -8865.688,E2 -8865.688} C_VEL
LIN {X 0,Y 447.107,Z 345.272,A -85,B 0,C 180,E1 -8866.861,E2 -8866.861} C_VEL
LIN {X 0,Y 446.617,Z 353.08,A -85,B 0,C 180,E1 -8868.026,E2 -8868.026} C_VEL
LIN {X 0,Y 446.229,Z 360.748,A -85,B 0,C 180,E1 -8869.439,E2 -8869.439} C_VEL
LIN {X 0,Y 445.861,Z 367.106,A -85,B 0,C 180,E1 -8870.912,E2 -8870.912} C_VEL
LIN {X 0,Y 445.601,Z 372.615,A -85,B 0,C 180,E1 -8872.611,E2 -8872.611} C_VEL
LIN {X 0,Y 445.382,Z 376.445,A -85,B 0,C 180,E1 -8874.278,E2 -8874.278} C_VEL
LIN {X 0,Y 445.299,Z 378.147,A -85,B 0,C 180,E1 -8875.377,E2 -8875.377} C_VEL
LIN {X 0,Y 445.224,Z 379.464,A -85,B 0,C 180,E1 -8876.786,E2 -8876.786} C_VEL
LIN {X 0,Y 445.24,Z 379.737,A -85,B 0,C 180,E1 -8878.607,E2 -8878.607} C_VEL
LIN {X 0,Y 445.327,Z 378.63,A -85,B 0,C 180,E1 -8880.227,E2 -8880.227} C_VEL
LIN {X 0,Y 445.441,Z 375.74,A -85,B 0,C 180,E1 -8882.074,E2 -8882.074} C_VEL
LIN {X 0,Y 445.656,Z 371.452,A -85,B 0,C 180,E1 -8883.796,E2 -8883.796} C_VEL
LIN {X 0,Y 445.902,Z 366.193,A -85,B 0,C 180,E1 -8885.312,E2 -8885.312} C_VEL
LIN {X 0,Y 446.233,Z 359.48,A -85,B 0,C 180,E1 -8886.812,E2 -8886.812} C_VEL
LIN {X 0,Y 446.607,Z 352.25,A -85,B 0,C 180,E1 -8888.102,E2 -8888.102} C_VEL
LIN {X 0,Y 446.109,Z 348.562,A -85,B 0,C 180,E1 -8888.693,E2 -8888.693} C_VEL
LIN {X 0,Y 443.638,Z 342.303,A -85,B 0,C 180,E1 -8889.635,E2 -8889.635} C_VEL
LIN {X 0,Y 441.256,Z 335.495,A -85,B 0,C 180,E1 -8890.515,E2 -8890.515} C_VEL
LIN {X 0,Y 440.89,Z 330.951,A -85,B 0,C 180,E1 -8891.001,E2 -8891.001} C_VEL
LIN {X 0,Y 441.498,Z 320.801,A -85,B 0,C 180,E1 -8891.916,E2 -8891.916} C_VEL
LIN {X 0,Y 442.031,Z 309.33,A -85,B 0,C 180,E1 -8892.743,E2 -8892.743} C_VEL
LIN {X 0,Y 442.502,Z 297.718,A -85,B 0,C 180,E1 -8893.388,E2 -8893.388} C_VEL
LIN {X 0,Y 442.912,Z 284.588,A -85,B 0,C 180,E1 -8893.907,E2 -8893.907} C_VEL
LIN {X 0,Y 443.238,Z 270.896,A -85,B 0,C 180,E1 -8894.244,E2 -8894.244} C_VEL
LIN {X 0,Y 444.167,Z 187.415,A -85,B 0,C 180,E1 -8895.628,E2 -8895.628} C_VEL
LIN {X 0,Y 440.693,Z 169.022,A -85,B 0,C 180,E1 -8896.107,E2 -8896.107} C_VEL
LIN {X 0,Y 441.098,Z 157.893,A -85,B 0,C 180,E1 -8898.512,E2 -8898.512} C_VEL
LIN {X 0,Y 439.508,Z 148.741,A -85,B 0,C 180,E1 -8900.624,E2 -8900.624} C_VEL
LIN {X 0,Y 439.564,Z 148.731,A -85,B 0,C 180,E1 -8903.574,E2 -8903.574} C_VEL
LIN {X 0,Y 439.422,Z 148.744,A -85,B 0,C 180,E1 -8905.413,E2 -8905.413} C_VEL
LIN {X 0,Y 439.635,Z 148.722,A -85,B 0,C 180,E1 -8908.168,E2 -8908.168} C_VEL
LIN {X 0,Y 439.713,Z 148.711,A -85,B 0,C 180,E1 -8910,E2 -8910} C_VEL
LIN {X 0,Y 439.609,Z 148.724,A -85,B 0,C 180,E1 -8912.749,E2 -8912.749} C_VEL
LIN {X 0,Y 439.562,Z 148.732,A -85,B 0,C 180,E1 -8916.426,E2 -8916.426} C_VEL
LIN {X 0,Y 439.493,Z 148.736,A -85,B 0,C 180,E1 -8919.202,E2 -8919.202} C_VEL
LIN {X 0,Y 439.468,Z 148.739,A -85,B 0,C 180,E1 -8922.938,E2 -8922.938} C_VEL
LIN {X 0,Y 439.405,Z 148.75,A -85,B 0,C 180,E1 -8926.328,E2 -8926.328} C_VEL
LIN {X 0,Y 439.404,Z 148.751,A -85,B 0,C 180,E1 -8929.626,E2 -8929.626} C_VEL
LIN {X 0,Y 439.366,Z 148.752,A -85,B 0,C 180,E1 -8932.576,E2 -8932.576} C_VEL
LIN {X 0,Y 439.369,Z 148.756,A -85,B 0,C 180,E1 -8935.587,E2 -8935.587} C_VEL
LIN {X 0,Y 439.392,Z 148.748,A -85,B 0,C 180,E1 -8938.676,E2 -8938.676} C_VEL
LIN {X 0,Y 439.369,Z 148.754,A -85,B 0,C 180,E1 -8942.03,E2 -8942.03} C_VEL
LIN {X 0,Y 439.393,Z 148.753,A -85,B 0,C 180,E1 -8945.34,E2 -8945.34} C_VEL
LIN {X 0,Y 439.365,Z 148.752,A -85,B 0,C 180,E1 -8948.597,E2 -8948.597} C_VEL
LIN {X 0,Y 439.351,Z 148.753,A -85,B 0,C 180,E1 -8952.21,E2 -8952.21} C_VEL
LIN {X 0,Y 439.4,Z 148.755,A -85,B 0,C 180,E1 -8955.27,E2 -8955.27} C_VEL
LIN {X 0,Y 439.356,Z 148.758,A -85,B 0,C 180,E1 -8959.016,E2 -8959.016} C_VEL
LIN {X 0,Y 439.37,Z 148.753,A -85,B 0,C 180,E1 -8961.609,E2 -8961.609} C_VEL
LIN {X 0,Y 439.398,Z 148.752,A -85,B 0,C 180,E1 -8964.844,E2 -8964.844} C_VEL
LIN {X 0,Y 439.369,Z 148.751,A -85,B 0,C 180,E1 -8968.139,E2 -8968.139} C_VEL
LIN {X 0,Y 439.403,Z 148.747,A -85,B 0,C 180,E1 -8971.606,E2 -8971.606} C_VEL
LIN {X 0,Y 439.369,Z 148.754,A -85,B 0,C 180,E1 -8974.413,E2 -8974.413} C_VEL
LIN {X 0,Y 439.364,Z 148.752,A -85,B 0,C 180,E1 -8977.424,E2 -8977.424} C_VEL
LIN {X 0,Y 439.444,Z 148.749,A -85,B 0,C 180,E1 -8980.664,E2 -8980.664} C_VEL
LIN {X 0,Y 439.422,Z 148.748,A -85,B 0,C 180,E1 -8984.223,E2 -8984.223} C_VEL
LIN {X 0,Y 439.489,Z 148.736,A -85,B 0,C 180,E1 -8987.285,E2 -8987.285} C_VEL
LIN {X 0,Y 439.487,Z 148.739,A -85,B 0,C 180,E1 -8990.798,E2 -8990.798} C_VEL
LIN {X 0,Y 439.562,Z 148.727,A -85,B 0,C 180,E1 -8993.574,E2 -8993.574} C_VEL
LIN {X 0,Y 439.408,Z 148.746,A -85,B 0,C 180,E1 -8995.413,E2 -8995.413} C_VEL
LIN {X 0,Y 439.631,Z 148.725,A -85,B 0,C 180,E1 -8998.168,E2 -8998.168} C_VEL
LIN {X 0,Y 439.673,Z 148.718,A -85,B 0,C 180,E1 -9000,E2 -9000} C_VEL
LIN {X 0,Y 439.606,Z 148.723,A -85,B 0,C 180,E1 -9002.749,E2 -9002.749} C_VEL
LIN {X 0,Y 439.562,Z 148.73,A -85,B 0,C 180,E1 -9006.426,E2 -9006.426} C_VEL
LIN {X 0,Y 439.478,Z 148.738,A -85,B 0,C 180,E1 -9009.202,E2 -9009.202} C_VEL
LIN {X 0,Y 439.455,Z 148.74,A -85,B 0,C 180,E1 -9012.938,E2 -9012.938} C_VEL
LIN {X 0,Y 439.4,Z 148.749,A -85,B 0,C 180,E1 -9016.325,E2 -9016.325} C_VEL
LIN {X 0,Y 439.372,Z 148.757,A -85,B 0,C 180,E1 -9019.628,E2 -9019.628} C_VEL
LIN {X 0,Y 439.355,Z 148.753,A -85,B 0,C 180,E1 -9022.576,E2 -9022.576} C_VEL
LIN {X 0,Y 439.357,Z 148.76,A -85,B 0,C 180,E1 -9025.588,E2 -9025.588} C_VEL
LIN {X 0,Y 439.379,Z 148.75,A -85,B 0,C 180,E1 -9028.676,E2 -9028.676} C_VEL
LIN {X 0,Y 439.345,Z 148.755,A -85,B 0,C 180,E1 -9032.024,E2 -9032.024} C_VEL
LIN {X 0,Y 439.386,Z 148.757,A -85,B 0,C 180,E1 -9035.338,E2 -9035.338} C_VEL
LIN {X 0,Y 439.353,Z 148.754,A -85,B 0,C 180,E1 -9038.598,E2 -9038.598} C_VEL
LIN {X 0,Y 439.364,Z 148.758,A -85,B 0,C 180,E1 -9041.253,E2 -9041.253} C_VEL
LIN {X 0,Y 439.398,Z 148.751,A -85,B 0,C 180,E1 -9044.73,E2 -9044.73} C_VEL
LIN {X 0,Y 439.347,Z 148.754,A -85,B 0,C 180,E1 -9047.789,E2 -9047.789} C_VEL
LIN {X 0,Y 439.36,Z 148.753,A -85,B 0,C 180,E1 -9050.22,E2 -9050.22} C_VEL
LIN {X 0,Y 439.365,Z 148.752,A -85,B 0,C 180,E1 -9053.712,E2 -9053.712} C_VEL
LIN {X 0,Y 439.343,Z 148.759,A -85,B 0,C 180,E1 -9057.051,E2 -9057.051} C_VEL
LIN {X 0,Y 439.358,Z 148.758,A -85,B 0,C 180,E1 -9060.272,E2 -9060.272} C_VEL
LIN {X 0,Y 439.36,Z 148.759,A -85,B 0,C 180,E1 -9063.509,E2 -9063.509} C_VEL
LIN {X 0,Y 441.738,Z 160.983,A -85,B 0,C 180,E1 -9066.065,E2 -9066.065} C_VEL
LIN {X 0,Y 441.823,Z 165.883,A -85,B 0,C 180,E1 -9067.027,E2 -9067.027} C_VEL
LIN {X 0,Y 440.887,Z 183.799,A -85,B 0,C 180,E1 -9070.442,E2 -9070.442} C_VEL
LIN {X 0,Y 440.442,Z 191.796,A -85,B 0,C 180,E1 -9071.939,E2 -9071.939} C_VEL
LIN {X 0,Y 443.885,Z 214.497,A -85,B 0,C 180,E1 -9072.463,E2 -9072.463} C_VEL
LIN {X 0,Y 443.029,Z 300.351,A -85,B 0,C 180,E1 -9073.912,E2 -9073.912} C_VEL
LIN {X 0,Y 442.569,Z 314.155,A -85,B 0,C 180,E1 -9074.338,E2 -9074.338} C_VEL
LIN {X 0,Y 442.02,Z 326.574,A -85,B 0,C 180,E1 -9074.909,E2 -9074.909} C_VEL
LIN {X 0,Y 441.458,Z 337.678,A -85,B 0,C 180,E1 -9075.596,E2 -9075.596} C_VEL
LIN {X 0,Y 440.78,Z 349.759,A -85,B 0,C 180,E1 -9076.56,E2 -9076.56} C_VEL
LIN {X 0,Y 440.199,Z 360.733,A -85,B 0,C 180,E1 -9077.67,E2 -9077.67} C_VEL
LIN {X 0,Y 439.55,Z 370.718,A -85,B 0,C 180,E1 -9078.938,E2 -9078.938} C_VEL
LIN {X 0,Y 439.067,Z 379.512,A -85,B 0,C 180,E1 -9080.324,E2 -9080.324} C_VEL
LIN {X 0,Y 438.738,Z 386.523,A -85,B 0,C 180,E1 -9081.711,E2 -9081.711} C_VEL
LIN {X 0,Y 438.493,Z 392.133,A -85,B 0,C 180,E1 -9083.096,E2 -9083.096} C_VEL
LIN {X 0,Y 438.373,Z 396.538,A -85,B 0,C 180,E1 -9084.48,E2 -9084.48} C_VEL
LIN {X 0,Y 438.339,Z 398.863,A -85,B 0,C 180,E1 -9085.402,E2 -9085.402} C_VEL
LIN {X 0,Y 438.279,Z 400.756,A -85,B 0,C 180,E1 -9086.322,E2 -9086.322} C_VEL
LIN {X 0,Y 438.34,Z 402.186,A -85,B 0,C 180,E1 -9087.243,E2 -9087.243} C_VEL
LIN {X 0,Y 438.253,Z 403.815,A -85,B 0,C 180,E1 -9089.081,E2 -9089.081} C_VEL
LIN {X 0,Y 438.255,Z 404.045,A -85,B 0,C 180,E1 -9090,E2 -9090} C_VEL
LIN {X 0,Y 438.253,Z 403.84,A -85,B 0,C 180,E1 -9090.919,E2 -9090.919} C_VEL
LIN {X 0,Y 438.34,Z 402.237,A -85,B 0,C 180,E1 -9092.757,E2 -9092.757} C_VEL
LIN {X 0,Y 438.279,Z 400.838,A -85,B 0,C 180,E1 -9093.678,E2 -9093.678} C_VEL
LIN {X 0,Y 438.38,Z 397.892,A -85,B 0,C 180,E1 -9095.059,E2 -9095.059} C_VEL
LIN {X 0,Y 438.448,Z 393.905,A -85,B 0,C 180,E1 -9096.443,E2 -9096.443} C_VEL
LIN {X 0,Y 438.682,Z 387.778,A -85,B 0,C 180,E1 -9098.058,E2 -9098.058} C_VEL
LIN {X 0,Y 439.031,Z 381.082,A -85,B 0,C 180,E1 -9099.444,E2 -9099.444} C_VEL
LIN {X 0,Y 439.467,Z 372.776,A -85,B 0,C 180,E1 -9100.831,E2 -9100.831} C_VEL
LIN {X 0,Y 440.066,Z 364.275,A -85,B 0,C 180,E1 -9101.983,E2 -9101.983} C_VEL
LIN {X 0,Y 440.688,Z 354.386,A -85,B 0,C 180,E1 -9103.075,E2 -9103.075} C_VEL
LIN {X 0,Y 441.275,Z 343.393,A -85,B 0,C 180,E1 -9104.057,E2 -9104.057} C_VEL
LIN {X 0,Y 441.877,Z 332.03,A -85,B 0,C 180,E1 -9104.861,E2 -9104.861} C_VEL
LIN {X 0,Y 442.495,Z 320.412,A -85,B 0,C 180,E1 -9105.488,E2 -9105.488} C_VEL
LIN {X 0,Y 443.02,Z 307.089,A -85,B 0,C 180,E1 -9106,E2 -9106} C_VEL
LIN {X 0,Y 443.419,Z 294.152,A -85,B 0,C 180,E1 -9106.31,E2 -9106.31} C_VEL
LIN {X 0,Y 444.129,Z 213.58,A -85,B 0,C 180,E1 -9107.662,E2 -9107.662} C_VEL
LIN {X 0,Y 440.49,Z 191.077,A -85,B 0,C 180,E1 -9108.236,E2 -9108.236} C_VEL
LIN {X 0,Y 441.339,Z 175.072,A -85,B 0,C 180,E1 -9111.24,E2 -9111.24} C_VEL
LIN {X 0,Y 441.968,Z 162.308,A -85,B 0,C 180,E1 -9113.673,E2 -9113.673} C_VEL
LIN {X 0,Y 439.833,Z 150.937,A -85,B 0,C 180,E1 -9116.034,E2 -9116.034} C_VEL
LIN {X 0,Y 439.35,Z 148.759,A -85,B 0,C 180,E1 -9116.531,E2 -9116.531} C_VEL
LIN {X 0,Y 439.358,Z 148.762,A -85,B 0,C 180,E1 -9119.728,E2 -9119.728} C_VEL
LIN {X 0,Y 439.343,Z 148.764,A -85,B 0,C 180,E1 -9122.949,E2 -9122.949} C_VEL
LIN {X 0,Y 439.364,Z 148.753,A -85,B 0,C 180,E1 -9126.289,E2 -9126.289} C_VEL
LIN {X 0,Y 439.348,Z 148.757,A -85,B 0,C 180,E1 -9128.599,E2 -9128.599} C_VEL
LIN {X 0,Y 439.346,Z 148.756,A -85,B 0,C 180,E1 -9132.211,E2 -9132.211} C_VEL
LIN {X 0,Y 439.398,Z 148.755,A -85,B 0,C 180,E1 -9135.27,E2 -9135.27} C_VEL
LIN {X 0,Y 439.35,Z 148.759,A -85,B 0,C 180,E1 -9139.016,E2 -9139.016} C_VEL
LIN {X 0,Y 439.334,Z 148.761,A -85,B 0,C 180,E1 -9142.563,E2 -9142.563} C_VEL
LIN {X 0,Y 439.389,Z 148.755,A -85,B 0,C 180,E1 -9144.843,E2 -9144.843} C_VEL
LIN {X 0,Y 439.348,Z 148.754,A -85,B 0,C 180,E1 -9148.137,E2 -9148.137} C_VEL
LIN {X 0,Y 439.379,Z 148.749,A -85,B 0,C 180,E1 -9151.324,E2 -9151.324} C_VEL
LIN {X 0,Y 439.353,Z 148.756,A -85,B 0,C 180,E1 -9154.412,E2 -9154.412} C_VEL
LIN {X 0,Y 439.352,Z 148.754,A -85,B 0,C 180,E1 -9157.424,E2 -9157.424} C_VEL
LIN {X 0,Y 439.384,Z 148.753,A -85,B 0,C 180,E1 -9160.686,E2 -9160.686} C_VEL
LIN {X 0,Y 439.404,Z 148.747,A -85,B 0,C 180,E1 -9164.222,E2 -9164.222} C_VEL
LIN {X 0,Y 439.469,Z 148.739,A -85,B 0,C 180,E1 -9167.297,E2 -9167.297} C_VEL
LIN {X 0,Y 439.476,Z 148.74,A -85,B 0,C 180,E1 -9170.798,E2 -9170.798} C_VEL
LIN {X 0,Y 439.557,Z 148.722,A -85,B 0,C 180,E1 -9173.574,E2 -9173.574} C_VEL
LIN {X 0,Y 439.405,Z 148.746,A -85,B 0,C 180,E1 -9175.413,E2 -9175.413} C_VEL
LIN {X 0,Y 439.63,Z 148.718,A -85,B 0,C 180,E1 -9178.168,E2 -9178.168} C_VEL
LIN {X 0,Y 439.673,Z 148.718,A -85,B 0,C 180,E1 -9180,E2 -9180} C_VEL
LIN {X 0,Y 439.606,Z 148.722,A -85,B 0,C 180,E1 -9182.749,E2 -9182.749} C_VEL
LIN {X 0,Y 439.562,Z 148.731,A -85,B 0,C 180,E1 -9186.426,E2 -9186.426} C_VEL
LIN {X 0,Y 439.479,Z 148.737,A -85,B 0,C 180,E1 -9189.202,E2 -9189.202} C_VEL
LIN {X 0,Y 439.469,Z 148.738,A -85,B 0,C 180,E1 -9192.938,E2 -9192.938} C_VEL
LIN {X 0,Y 439.401,Z 148.751,A -85,B 0,C 180,E1 -9196.326,E2 -9196.326} C_VEL
LIN {X 0,Y 439.381,Z 148.757,A -85,B 0,C 180,E1 -9199.627,E2 -9199.627} C_VEL
LIN {X 0,Y 439.363,Z 148.754,A -85,B 0,C 180,E1 -9202.576,E2 -9202.576} C_VEL
LIN {X 0,Y 439.37,Z 148.76,A -85,B 0,C 180,E1 -9205.587,E2 -9205.587} C_VEL
LIN {X 0,Y 439.384,Z 148.753,A -85,B 0,C 180,E1 -9208.676,E2 -9208.676} C_VEL
LIN {X 0,Y 439.369,Z 148.758,A -85,B 0,C 180,E1 -9212.029,E2 -9212.029} C_VEL
LIN {X 0,Y 439.418,Z 148.94,A -85,B 0,C 180,E1 -9215.442,E2 -9215.442} C_VEL
LIN {X 0,Y 441.179,Z 158.268,A -85,B 0,C 180,E1 -9217.541,E2 -9217.541} C_VEL
LIN {X 0,Y 440.908,Z 169.478,A -85,B 0,C 180,E1 -9219.865,E2 -9219.865} C_VEL
LIN {X 0,Y 444.462,Z 187.467,A -85,B 0,C 180,E1 -9220.337,E2 -9220.337} C_VEL
LIN {X 0,Y 443.358,Z 277.169,A -85,B 0,C 180,E1 -9221.859,E2 -9221.859} C_VEL
LIN {X 0,Y 443.015,Z 290.764,A -85,B 0,C 180,E1 -9222.286,E2 -9222.286} C_VEL
LIN {X 0,Y 442.615,Z 302.496,A -85,B 0,C 180,E1 -9222.829,E2 -9222.829} C_VEL
LIN {X 0,Y 441.983,Z 314.511,A -85,B 0,C 180,E1 -9223.573,E2 -9223.573} C_VEL
LIN {X 0,Y 441.313,Z 326.753,A -85,B 0,C 180,E1 -9224.564,E2 -9224.564} C_VEL
LIN {X 0,Y 440.715,Z 336.695,A -85,B 0,C 180,E1 -9225.576,E2 -9225.576} C_VEL
LIN {X 0,Y 440.079,Z 346.54,A -85,B 0,C 180,E1 -9226.825,E2 -9226.825} C_VEL
LIN {X 0,Y 439.564,Z 354.56,A -85,B 0,C 180,E1 -9228.076,E2 -9228.076} C_VEL
LIN {X 0,Y 439.099,Z 362.369,A -85,B 0,C 180,E1 -9229.592,E2 -9229.592} C_VEL
LIN {X 0,Y 438.813,Z 367.284,A -85,B 0,C 180,E1 -9230.783,E2 -9230.783} C_VEL
LIN {X 0,Y 438.536,Z 372.727,A -85,B 0,C 180,E1 -9232.483,E2 -9232.483} C_VEL
LIN {X 0,Y 438.316,Z 376.585,A -85,B 0,C 180,E1 -9234.179,E2 -9234.179} C_VEL
LIN {X 0,Y 438.175,Z 378.958,A -85,B 0,C 180,E1 -9235.849,E2 -9235.849} C_VEL
LIN {X 0,Y 438.124,Z 379.758,A -85,B 0,C 180,E1 -9236.948,E2 -9236.948} C_VEL
LIN {X 0,Y 438.146,Z 380.001,A -85,B 0,C 180,E1 -9238.227,E2 -9238.227} C_VEL
LIN {X 0,Y 438.213,Z 379.056,A -85,B 0,C 180,E1 -9240.003,E2 -9240.003} C_VEL
LIN {X 0,Y 438.333,Z 376.445,A -85,B 0,C 180,E1 -9241.866,E2 -9241.866} C_VEL
LIN {X 0,Y 438.499,Z 373.142,A -85,B 0,C 180,E1 -9243.335,E2 -9243.335} C_VEL
LIN {X 0,Y 438.751,Z 368.372,A -85,B 0,C 180,E1 -9244.882,E2 -9244.882} C_VEL
LIN {X 0,Y 439.033,Z 362.227,A -85,B 0,C 180,E1 -9246.409,E2 -9246.409} C_VEL
LIN {X 0,Y 439.402,Z 355.259,A -85,B 0,C 180,E1 -9247.775,E2 -9247.775} C_VEL
LIN {X 0,Y 439.961,Z 346.283,A -85,B 0,C 180,E1 -9249.18,E2 -9249.18} C_VEL
LIN {X 0,Y 440.587,Z 336.373,A -85,B 0,C 180,E1 -9250.428,E2 -9250.428} C_VEL
LIN {X 0,Y 440.89,Z 330.951,A -85,B 0,C 180,E1 -9251.001,E2 -9251.001} C_VEL
LIN {X 0,Y 440.519,Z 326.319,A -85,B 0,C 180,E1 -9251.464,E2 -9251.464} C_VEL
LIN {X 0,Y 438.149,Z 318.57,A -85,B 0,C 180,E1 -9252.209,E2 -9252.209} C_VEL
LIN {X 0,Y 435.762,Z 310.423,A -85,B 0,C 180,E1 -9252.885,E2 -9252.885} C_VEL
LIN {X 0,Y 435.343,Z 305.108,A -85,B 0,C 180,E1 -9253.234,E2 -9253.234} C_VEL
LIN {X 0,Y 435.783,Z 292.905,A -85,B 0,C 180,E1 -9253.847,E2 -9253.847} C_VEL
LIN {X 0,Y 436.246,Z 280.139,A -85,B 0,C 180,E1 -9254.285,E2 -9254.285} C_VEL
LIN {X 0,Y 436.467,Z 262.138,A -85,B 0,C 180,E1 -9254.642,E2 -9254.642} C_VEL
LIN {X 0,Y 437.334,Z 187.965,A -85,B 0,C 180,E1 -9255.891,E2 -9255.891} C_VEL
LIN {X 0,Y 433.743,Z 169.301,A -85,B 0,C 180,E1 -9256.368,E2 -9256.368} C_VEL
LIN {X 0,Y 434.143,Z 159.287,A -85,B 0,C 180,E1 -9258.562,E2 -9258.562} C_VEL
LIN {X 0,Y 432.465,Z 149.618,A -85,B 0,C 180,E1 -9260.824,E2 -9260.824} C_VEL
LIN {X 0,Y 432.52,Z 149.609,A -85,B 0,C 180,E1 -9263.469,E2 -9263.469} C_VEL
LIN {X 0,Y 432.39,Z 149.621,A -85,B 0,C 180,E1 -9265.338,E2 -9265.338} C_VEL
LIN {X 0,Y 432.604,Z 149.598,A -85,B 0,C 180,E1 -9268.138,E2 -9268.138} C_VEL
LIN {X 0,Y 432.663,Z 149.589,A -85,B 0,C 180,E1 -9270,E2 -9270} C_VEL
LIN {X 0,Y 432.562,Z 149.601,A -85,B 0,C 180,E1 -9272.794,E2 -9272.794} C_VEL
LIN {X 0,Y 432.575,Z 149.598,A -85,B 0,C 180,E1 -9275.594,E2 -9275.594} C_VEL
LIN {X 0,Y 432.465,Z 149.616,A -85,B 0,C 180,E1 -9278.41,E2 -9278.41} C_VEL
LIN {X 0,Y 432.462,Z 149.618,A -85,B 0,C 180,E1 -9282.197,E2 -9282.197} C_VEL
LIN {X 0,Y 432.391,Z 149.627,A -85,B 0,C 180,E1 -9286.04,E2 -9286.04} C_VEL
LIN {X 0,Y 432.389,Z 149.623,A -85,B 0,C 180,E1 -9289.485,E2 -9289.485} C_VEL
LIN {X 0,Y 432.315,Z 149.63,A -85,B 0,C 180,E1 -9292.965,E2 -9292.965} C_VEL
LIN {X 0,Y 432.32,Z 149.633,A -85,B 0,C 180,E1 -9296.036,E2 -9296.036} C_VEL
LIN {X 0,Y 432.329,Z 149.63,A -85,B 0,C 180,E1 -9299.189,E2 -9299.189} C_VEL
LIN {X 0,Y 432.324,Z 149.629,A -85,B 0,C 180,E1 -9302.443,E2 -9302.443} C_VEL
LIN {X 0,Y 432.339,Z 149.631,A -85,B 0,C 180,E1 -9305.818,E2 -9305.818} C_VEL
LIN {X 0,Y 432.328,Z 149.629,A -85,B 0,C 180,E1 -9308.712,E2 -9308.712} C_VEL
LIN {X 0,Y 432.306,Z 149.633,A -85,B 0,C 180,E1 -9311.801,E2 -9311.801} C_VEL
LIN {X 0,Y 432.336,Z 149.627,A -85,B 0,C 180,E1 -9314.348,E2 -9314.348} C_VEL
LIN {X 0,Y 432.305,Z 149.636,A -85,B 0,C 180,E1 -9317.018,E2 -9317.018} C_VEL
LIN {X 0,Y 432.31,Z 149.631,A -85,B 0,C 180,E1 -9319.825,E2 -9319.825} C_VEL
LIN {X 0,Y 432.308,Z 149.637,A -85,B 0,C 180,E1 -9323.022,E2 -9323.022} C_VEL
LIN {X 0,Y 432.336,Z 149.627,A -85,B 0,C 180,E1 -9326.002,E2 -9326.002} C_VEL
LIN {X 0,Y 432.344,Z 149.628,A -85,B 0,C 180,E1 -9329.491,E2 -9329.491} C_VEL
LIN {X 0,Y 432.338,Z 149.627,A -85,B 0,C 180,E1 -9331.873,E2 -9331.873} C_VEL
LIN {X 0,Y 432.327,Z 149.633,A -85,B 0,C 180,E1 -9334.997,E2 -9334.997} C_VEL
LIN {X 0,Y 432.358,Z 149.625,A -85,B 0,C 180,E1 -9338.046,E2 -9338.046} C_VEL
LIN {X 0,Y 432.384,Z 149.624,A -85,B 0,C 180,E1 -9341.029,E2 -9341.029} C_VEL
LIN {X 0,Y 432.392,Z 149.621,A -85,B 0,C 180,E1 -9343.96,E2 -9343.96} C_VEL
LIN {X 0,Y 432.463,Z 149.612,A -85,B 0,C 180,E1 -9347.803,E2 -9347.803} C_VEL
LIN {X 0,Y 432.452,Z 149.613,A -85,B 0,C 180,E1 -9351.589,E2 -9351.589} C_VEL
LIN {X 0,Y 432.574,Z 149.604,A -85,B 0,C 180,E1 -9354.406,E2 -9354.406} C_VEL
LIN {X 0,Y 432.6,Z 149.601,A -85,B 0,C 180,E1 -9358.138,E2 -9358.138} C_VEL
LIN {X 0,Y 432.624,Z 149.596,A -85,B 0,C 180,E1 -9360,E2 -9360} C_VEL
LIN {X 0,Y 432.56,Z 149.6,A -85,B 0,C 180,E1 -9362.794,E2 -9362.794} C_VEL
LIN {X 0,Y 432.518,Z 149.606,A -85,B 0,C 180,E1 -9366.531,E2 -9366.531} C_VEL
LIN {X 0,Y 432.424,Z 149.617,A -85,B 0,C 180,E1 -9369.354,E2 -9369.354} C_VEL
LIN {X 0,Y 432.422,Z 149.616,A -85,B 0,C 180,E1 -9372.795,E2 -9372.795} C_VEL
LIN {X 0,Y 432.359,Z 149.625,A -85,B 0,C 180,E1 -9376.453,E2 -9376.453} C_VEL
LIN {X 0,Y 432.305,Z 149.635,A -85,B 0,C 180,E1 -9379.962,E2 -9379.962} C_VEL
LIN {X 0,Y 432.304,Z 149.632,A -85,B 0,C 180,E1 -9382.965,E2 -9382.965} C_VEL
LIN {X 0,Y 432.308,Z 149.633,A -85,B 0,C 180,E1 -9386.036,E2 -9386.036} C_VEL
LIN {X 0,Y 432.317,Z 149.633,A -85,B 0,C 180,E1 -9389.189,E2 -9389.189} C_VEL
LIN {X 0,Y 432.307,Z 149.631,A -85,B 0,C 180,E1 -9392.444,E2 -9392.444} C_VEL
LIN {X 0,Y 432.334,Z 149.629,A -85,B 0,C 180,E1 -9395.818,E2 -9395.818} C_VEL
LIN {X 0,Y 432.301,Z 149.638,A -85,B 0,C 180,E1 -9399.348,E2 -9399.348} C_VEL
LIN {X 0,Y 432.304,Z 149.632,A -85,B 0,C 180,E1 -9401.801,E2 -9401.801} C_VEL
LIN {X 0,Y 432.335,Z 149.628,A -85,B 0,C 180,E1 -9404.347,E2 -9404.347} C_VEL
LIN {X 0,Y 432.302,Z 149.639,A -85,B 0,C 180,E1 -9407.019,E2 -9407.019} C_VEL
LIN {X 0,Y 432.289,Z 149.633,A -85,B 0,C 180,E1 -9409.828,E2 -9409.828} C_VEL
LIN {X 0,Y 432.296,Z 149.638,A -85,B 0,C 180,E1 -9413.021,E2 -9413.021} C_VEL
LIN {X 0,Y 432.331,Z 149.628,A -85,B 0,C 180,E1 -9416.002,E2 -9416.002} C_VEL
LIN {X 0,Y 432.332,Z 149.631,A -85,B 0,C 180,E1 -9419.494,E2 -9419.494} C_VEL
LIN {X 0,Y 432.313,Z 149.634,A -85,B 0,C 180,E1 -9421.872,E2 -9421.872} C_VEL
LIN {X 0,Y 432.326,Z 149.793,A -85,B 0,C 180,E1 -9423.314,E2 -9423.314} C_VEL
LIN {X 0,Y 434.733,Z 161.986,A -85,B 0,C 180,E1 -9425.908,E2 -9425.908} C_VEL
LIN {X 0,Y 434.954,Z 166.064,A -85,B 0,C 180,E1 -9426.73,E2 -9426.73} C_VEL
LIN {X 0,Y 433.907,Z 184.811,A -85,B 0,C 180,E1 -9430.361,E2 -9430.361} C_VEL
LIN {X 0,Y 433.472,Z 191.54,A -85,B 0,C 180,E1 -9431.648,E2 -9431.648} C_VEL
LIN {X 0,Y 437.087,Z 215.208,A -85,B 0,C 180,E1 -9432.211,E2 -9432.211} C_VEL
LIN {X 0,Y 436.215,Z 299.562,A -85,B 0,C 180,E1 -9433.653,E2 -9433.653} C_VEL
LIN {X 0,Y 435.789,Z 312.801,A -85,B 0,C 180,E1 -9434.058,E2 -9434.058} C_VEL
LIN {X 0,Y 435.145,Z 326.095,A -85,B 0,C 180,E1 -9434.664,E2 -9434.664} C_VEL
LIN {X 0,Y 434.552,Z 337.274,A -85,B 0,C 180,E1 -9435.362,E2 -9435.362} C_VEL
LIN {X 0,Y 433.909,Z 348.318,A -85,B 0,C 180,E1 -9436.244,E2 -9436.244} C_VEL
LIN {X 0,Y 433.233,Z 359.369,A -85,B 0,C 180,E1 -9437.35,E2 -9437.35} C_VEL
LIN {X 0,Y 432.713,Z 368.789,A -85,B 0,C 180,E1 -9438.524,E2 -9438.524} C_VEL
LIN {X 0,Y 432.163,Z 376.514,A -85,B 0,C 180,E1 -9439.695,E2 -9439.695} C_VEL
LIN {X 0,Y 431.793,Z 384.081,A -85,B 0,C 180,E1 -9441.105,E2 -9441.105} C_VEL
LIN {X 0,Y 431.49,Z 390.159,A -85,B 0,C 180,E1 -9442.513,E2 -9442.513} C_VEL
LIN {X 0,Y 431.268,Z 395.335,A -85,B 0,C 180,E1 -9444.04,E2 -9444.04} C_VEL
LIN {X 0,Y 431.268,Z 398.645,A -85,B 0,C 180,E1 -9445.326,E2 -9445.326} C_VEL
LIN {X 0,Y 431.186,Z 400.541,A -85,B 0,C 180,E1 -9446.262,E2 -9446.262} C_VEL
LIN {X 0,Y 431.236,Z 401.979,A -85,B 0,C 180,E1 -9447.198,E2 -9447.198} C_VEL
LIN {X 0,Y 431.203,Z 402.993,A -85,B 0,C 180,E1 -9448.132,E2 -9448.132} C_VEL
LIN {X 0,Y 431.169,Z 403.849,A -85,B 0,C 180,E1 -9450,E2 -9450} C_VEL
LIN {X 0,Y 431.17,Z 403.65,A -85,B 0,C 180,E1 -9450.934,E2 -9450.934} C_VEL
LIN {X 0,Y 431.203,Z 403.047,A -85,B 0,C 180,E1 -9451.868,E2 -9451.868} C_VEL
LIN {X 0,Y 431.235,Z 402.052,A -85,B 0,C 180,E1 -9452.802,E2 -9452.802} C_VEL
LIN {X 0,Y 431.186,Z 400.656,A -85,B 0,C 180,E1 -9453.738,E2 -9453.738} C_VEL
LIN {X 0,Y 431.29,Z 397.716,A -85,B 0,C 180,E1 -9455.142,E2 -9455.142} C_VEL
LIN {X 0,Y 431.376,Z 393.735,A -85,B 0,C 180,E1 -9456.549,E2 -9456.549} C_VEL
LIN {X 0,Y 431.623,Z 387.62,A -85,B 0,C 180,E1 -9458.191,E2 -9458.191} C_VEL
LIN {X 0,Y 431.981,Z 380.93,A -85,B 0,C 180,E1 -9459.6,E2 -9459.6} C_VEL
LIN {X 0,Y 432.451,Z 372.631,A -85,B 0,C 180,E1 -9461.009,E2 -9461.009} C_VEL
LIN {X 0,Y 433.104,Z 364.144,A -85,B 0,C 180,E1 -9462.178,E2 -9462.178} C_VEL
LIN {X 0,Y 433.736,Z 353.391,A -85,B 0,C 180,E1 -9463.378,E2 -9463.378} C_VEL
LIN {X 0,Y 434.466,Z 341.889,A -85,B 0,C 180,E1 -9464.401,E2 -9464.401} C_VEL
LIN {X 0,Y 435.117,Z 330.103,A -85,B 0,C 180,E1 -9465.217,E2 -9465.217} C_VEL
LIN {X 0,Y 435.813,Z 317.878,A -85,B 0,C 180,E1 -9465.851,E2 -9465.851} C_VEL
LIN {X 0,Y 436.307,Z 305.457,A -85,B 0,C 180,E1 -9466.313,E2 -9466.313} C_VEL
LIN {X 0,Y 436.614,Z 293.055,A -85,B 0,C 180,E1 -9466.602,E2 -9466.602} C_VEL
LIN {X 0,Y 437.418,Z 214.61,A -85,B 0,C 180,E1 -9467.936,E2 -9467.936} C_VEL
LIN {X 0,Y 433.556,Z 190.888,A -85,B 0,C 180,E1 -9468.549,E2 -9468.549} C_VEL
LIN {X 0,Y 434.54,Z 173.682,A -85,B 0,C 180,E1 -9471.839,E2 -9471.839} C_VEL
LIN {X 0,Y 435.039,Z 163.48,A -85,B 0,C 180,E1 -9473.821,E2 -9473.821} C_VEL
LIN {X 0,Y 433.09,Z 153.228,A -85,B 0,C 180,E1 -9475.986,E2 -9475.986} C_VEL
LIN {X 0,Y 432.308,Z 149.638,A -85,B 0,C 180,E1 -9476.793,E2 -9476.793} C_VEL
LIN {X 0,Y 432.316,Z 149.639,A -85,B 0,C 180,E1 -9479.19,E2 -9479.19} C_VEL
LIN {X 0,Y 432.306,Z 149.638,A -85,B 0,C 180,E1 -9482.445,E2 -9482.445} C_VEL
LIN {X 0,Y 432.331,Z 149.631,A -85,B 0,C 180,E1 -9485.819,E2 -9485.819} C_VEL
LIN {X 0,Y 432.313,Z 149.635,A -85,B 0,C 180,E1 -9488.71,E2 -9488.71} C_VEL
LIN {X 0,Y 432.302,Z 149.634,A -85,B 0,C 180,E1 -9491.801,E2 -9491.801} C_VEL
LIN {X 0,Y 432.334,Z 149.631,A -85,B 0,C 180,E1 -9494.348,E2 -9494.348} C_VEL
LIN {X 0,Y 432.302,Z 149.636,A -85,B 0,C 180,E1 -9497.019,E2 -9497.019} C_VEL
LIN {X 0,Y 432.289,Z 149.631,A -85,B 0,C 180,E1 -9499.828,E2 -9499.828} C_VEL
LIN {X 0,Y 432.295,Z 149.634,A -85,B 0,C 180,E1 -9503.021,E2 -9503.021} C_VEL
LIN {X 0,Y 432.332,Z 149.628,A -85,B 0,C 180,E1 -9506.003,E2 -9506.003} C_VEL
LIN {X 0,Y 432.333,Z 149.628,A -85,B 0,C 180,E1 -9509.494,E2 -9509.494} C_VEL
LIN {X 0,Y 432.315,Z 149.628,A -85,B 0,C 180,E1 -9511.872,E2 -9511.872} C_VEL
LIN {X 0,Y 432.315,Z 149.628,A -85,B 0,C 180,E1 -9514.996,E2 -9514.996} C_VEL
LIN {X 0,Y 432.351,Z 149.628,A -85,B 0,C 180,E1 -9518.045,E2 -9518.045} C_VEL
LIN {X 0,Y 432.34,Z 149.629,A -85,B 0,C 180,E1 -9521.027,E2 -9521.027} C_VEL
LIN {X 0,Y 432.359,Z 149.624,A -85,B 0,C 180,E1 -9523.958,E2 -9523.958} C_VEL
LIN {X 0,Y 432.451,Z 149.614,A -85,B 0,C 180,E1 -9527.803,E2 -9527.803} C_VEL
LIN {X 0,Y 432.449,Z 149.613,A -85,B 0,C 180,E1 -9531.589,E2 -9531.589} C_VEL
LIN {X 0,Y 432.551,Z 149.602,A -85,B 0,C 180,E1 -9534.406,E2 -9534.406} C_VEL
LIN {X 0,Y 432.599,Z 149.594,A -85,B 0,C 180,E1 -9538.138,E2 -9538.138} C_VEL
LIN {X 0,Y 432.624,Z 149.596,A -85,B 0,C 180,E1 -9540,E2 -9540} C_VEL
LIN {X 0,Y 432.56,Z 149.6,A -85,B 0,C 180,E1 -9542.794,E2 -9542.794} C_VEL
LIN {X 0,Y 432.519,Z 149.607,A -85,B 0,C 180,E1 -9546.531,E2 -9546.531} C_VEL
LIN {X 0,Y 432.424,Z 149.616,A -85,B 0,C 180,E1 -9549.354,E2 -9549.354} C_VEL
LIN {X 0,Y 432.435,Z 149.614,A -85,B 0,C 180,E1 -9552.803,E2 -9552.803} C_VEL
LIN {X 0,Y 432.36,Z 149.627,A -85,B 0,C 180,E1 -9556.453,E2 -9556.453} C_VEL
LIN {X 0,Y 432.317,Z 149.634,A -85,B 0,C 180,E1 -9559.962,E2 -9559.962} C_VEL
LIN {X 0,Y 432.313,Z 149.633,A -85,B 0,C 180,E1 -9562.965,E2 -9562.965} C_VEL
LIN {X 0,Y 432.321,Z 149.636,A -85,B 0,C 180,E1 -9566.035,E2 -9566.035} C_VEL
LIN {X 0,Y 432.325,Z 149.635,A -85,B 0,C 180,E1 -9569.189,E2 -9569.189} C_VEL
LIN {X 0,Y 432.325,Z 149.634,A -85,B 0,C 180,E1 -9572.443,E2 -9572.443} C_VEL
LIN {X 0,Y 432.376,Z 149.645,A -85,B 0,C 180,E1 -9575.152,E2 -9575.152} C_VEL
LIN {X 0,Y 434.285,Z 160.067,A -85,B 0,C 180,E1 -9577.536,E2 -9577.536} C_VEL
LIN {X 0,Y 433.97,Z 169.509,A -85,B 0,C 180,E1 -9579.543,E2 -9579.543} C_VEL
LIN {X 0,Y 437.737,Z 188.182,A -85,B 0,C 180,E1 -9580.05,E2 -9580.05} C_VEL
LIN {X 0,Y 436.58,Z 276.998,A -85,B 0,C 180,E1 -9581.578,E2 -9581.578} C_VEL
LIN {X 0,Y 436.22,Z 290.439,A -85,B 0,C 180,E1 -9582.001,E2 -9582.001} C_VEL
LIN {X 0,Y 435.786,Z 303.037,A -85,B 0,C 180,E1 -9582.59,E2 -9582.59} C_VEL
LIN {X 0,Y 435.115,Z 315.369,A -85,B 0,C 180,E1 -9583.377,E2 -9583.377} C_VEL
LIN {X 0,Y 434.449,Z 326.864,A -85,B 0,C 180,E1 -9584.327,E2 -9584.327} C_VEL
LIN {X 0,Y 433.821,Z 336.489,A -85,B 0,C 180,E1 -9585.317,E2 -9585.317} C_VEL
LIN {X 0,Y 433.161,Z 346.178,A -85,B 0,C 180,E1 -9586.551,E2 -9586.551} C_VEL
LIN {X 0,Y 432.562,Z 354.832,A -85,B 0,C 180,E1 -9587.917,E2 -9587.917} C_VEL
LIN {X 0,Y 432.101,Z 362.433,A -85,B 0,C 180,E1 -9589.414,E2 -9589.414} C_VEL
LIN {X 0,Y 431.686,Z 368.811,A -85,B 0,C 180,E1 -9591.034,E2 -9591.034} C_VEL
LIN {X 0,Y 431.471,Z 372.845,A -85,B 0,C 180,E1 -9592.351,E2 -9592.351} C_VEL
LIN {X 0,Y 431.256,Z 376.73,A -85,B 0,C 180,E1 -9594.078,E2 -9594.078} C_VEL
LIN {X 0,Y 431.104,Z 378.469,A -85,B 0,C 180,E1 -9595.209,E2 -9595.209} C_VEL
LIN {X 0,Y 431.055,Z 379.605,A -85,B 0,C 180,E1 -9596.334,E2 -9596.334} C_VEL
LIN {X 0,Y 431.039,Z 380.23,A -85,B 0,C 180,E1 -9597.979,E2 -9597.979} C_VEL
LIN {X 0,Y 431.104,Z 379.469,A -85,B 0,C 180,E1 -9599.772,E2 -9599.772} C_VEL
LIN {X 0,Y 431.143,Z 378.479,A -85,B 0,C 180,E1 -9600.723,E2 -9600.723} C_VEL
LIN {X 0,Y 431.29,Z 375.849,A -85,B 0,C 180,E1 -9602.327,E2 -9602.327} C_VEL
LIN {X 0,Y 431.49,Z 371.988,A -85,B 0,C 180,E1 -9603.911,E2 -9603.911} C_VEL
LIN {X 0,Y 431.773,Z 367.14,A -85,B 0,C 180,E1 -9605.379,E2 -9605.379} C_VEL
LIN {X 0,Y 432.089,Z 361.311,A -85,B 0,C 180,E1 -9606.769,E2 -9606.769} C_VEL
LIN {X 0,Y 432.542,Z 353.209,A -85,B 0,C 180,E1 -9608.306,E2 -9608.306} C_VEL
LIN {X 0,Y 433.116,Z 344.82,A -85,B 0,C 180,E1 -9609.581,E2 -9609.581} C_VEL
LIN {X 0,Y 433.705,Z 335.591,A -85,B 0,C 180,E1 -9610.721,E2 -9610.721} C_VEL
LIN {X 0,Y 434.362,Z 324.222,A -85,B 0,C 180,E1 -9611.852,E2 -9611.852} C_VEL
LIN {X 0,Y 435,Z 312.678,A -85,B 0,C 180,E1 -9612.756,E2 -9612.756} C_VEL
LIN {X 0,Y 435.343,Z 305.108,A -85,B 0,C 180,E1 -9613.234,E2 -9613.234} C_VEL
LIN {X 0,Y 434.923,Z 299.725,A -85,B 0,C 180,E1 -9613.555,E2 -9613.555} C_VEL
LIN {X 0,Y 432.471,Z 290.898,A -85,B 0,C 180,E1 -9614.064,E2 -9614.064} C_VEL
LIN {X 0,Y 429.97,Z 281.836,A -85,B 0,C 180,E1 -9614.477,E2 -9614.477} C_VEL
LIN {X 0,Y 429.463,Z 276.095,A -85,B 0,C 180,E1 -9614.643,E2 -9614.643} C_VEL
LIN {X 0,Y 430.509,Z 188.564,A -85,B 0,C 180,E1 -9616.161,E2 -9616.161} C_VEL
LIN {X 0,Y 426.805,Z 169.432,A -85,B 0,C 180,E1 -9616.671,E2 -9616.671} C_VEL
LIN {X 0,Y 427.188,Z 160.683,A -85,B 0,C 180,E1 -9618.614,E2 -9618.614} C_VEL
LIN {X 0,Y 425.436,Z 150.493,A -85,B 0,C 180,E1 -9621.061,E2 -9621.061} C_VEL
LIN {X 0,Y 425.533,Z 150.481,A -85,B 0,C 180,E1 -9624.313,E2 -9624.313} C_VEL
LIN {X 0,Y 425.574,Z 150.473,A -85,B 0,C 180,E1 -9628.107,E2 -9628.107} C_VEL
LIN {X 0,Y 425.511,Z 150.479,A -85,B 0,C 180,E1 -9630.946,E2 -9630.946} C_VEL
LIN {X 0,Y 425.518,Z 150.478,A -85,B 0,C 180,E1 -9632.84,E2 -9632.84} C_VEL
LIN {X 0,Y 425.529,Z 150.477,A -85,B 0,C 180,E1 -9635.687,E2 -9635.687} C_VEL
LIN {X 0,Y 425.409,Z 150.493,A -85,B 0,C 180,E1 -9638.551,E2 -9638.551} C_VEL
LIN {X 0,Y 425.415,Z 150.493,A -85,B 0,C 180,E1 -9642.402,E2 -9642.402} C_VEL
LIN {X 0,Y 425.307,Z 150.504,A -85,B 0,C 180,E1 -9645.331,E2 -9645.331} C_VEL
LIN {X 0,Y 425.316,Z 150.505,A -85,B 0,C 180,E1 -9648.298,E2 -9648.298} C_VEL
LIN {X 0,Y 425.295,Z 150.506,A -85,B 0,C 180,E1 -9651.319,E2 -9651.319} C_VEL
LIN {X 0,Y 425.302,Z 150.504,A -85,B 0,C 180,E1 -9654.651,E2 -9654.651} C_VEL
LIN {X 0,Y 425.254,Z 150.515,A -85,B 0,C 180,E1 -9657.565,E2 -9657.565} C_VEL
LIN {X 0,Y 425.293,Z 150.505,A -85,B 0,C 180,E1 -9660.761,E2 -9660.761} C_VEL
LIN {X 0,Y 425.294,Z 150.505,A -85,B 0,C 180,E1 -9664.284,E2 -9664.284} C_VEL
LIN {X 0,Y 425.278,Z 150.511,A -85,B 0,C 180,E1 -9667.695,E2 -9667.695} C_VEL
LIN {X 0,Y 425.246,Z 150.51,A -85,B 0,C 180,E1 -9670.515,E2 -9670.515} C_VEL
LIN {X 0,Y 425.249,Z 150.517,A -85,B 0,C 180,E1 -9673.349,E2 -9673.349} C_VEL
LIN {X 0,Y 425.259,Z 150.509,A -85,B 0,C 180,E1 -9676.044,E2 -9676.044} C_VEL
LIN {X 0,Y 425.256,Z 150.513,A -85,B 0,C 180,E1 -9679.484,E2 -9679.484} C_VEL
LIN {X 0,Y 425.279,Z 150.507,A -85,B 0,C 180,E1 -9682.489,E2 -9682.489} C_VEL
LIN {X 0,Y 425.289,Z 150.505,A -85,B 0,C 180,E1 -9685.815,E2 -9685.815} C_VEL
LIN {X 0,Y 425.291,Z 150.508,A -85,B 0,C 180,E1 -9689.24,E2 -9689.24} C_VEL
LIN {X 0,Y 425.263,Z 150.511,A -85,B 0,C 180,E1 -9692.436,E2 -9692.436} C_VEL
LIN {X 0,Y 425.327,Z 150.501,A -85,B 0,C 180,E1 -9695.6,E2 -9695.6} C_VEL
LIN {X 0,Y 425.293,Z 150.512,A -85,B 0,C 180,E1 -9698.681,E2 -9698.681} C_VEL
LIN {X 0,Y 425.316,Z 150.502,A -85,B 0,C 180,E1 -9701.702,E2 -9701.702} C_VEL
LIN {X 0,Y 425.306,Z 150.509,A -85,B 0,C 180,E1 -9704.669,E2 -9704.669} C_VEL
LIN {X 0,Y 425.416,Z 150.489,A -85,B 0,C 180,E1 -9707.598,E2 -9707.598} C_VEL
LIN {X 0,Y 425.401,Z 150.491,A -85,B 0,C 180,E1 -9711.449,E2 -9711.449} C_VEL
LIN {X 0,Y 425.529,Z 150.483,A -85,B 0,C 180,E1 -9714.313,E2 -9714.313} C_VEL
LIN {X 0,Y 425.569,Z 150.476,A -85,B 0,C 180,E1 -9718.107,E2 -9718.107} C_VEL
LIN {X 0,Y 425.576,Z 150.474,A -85,B 0,C 180,E1 -9720,E2 -9720} C_VEL
LIN {X 0,Y 425.515,Z 150.477,A -85,B 0,C 180,E1 -9722.84,E2 -9722.84} C_VEL
LIN {X 0,Y 425.479,Z 150.482,A -85,B 0,C 180,E1 -9726.64,E2 -9726.64} C_VEL
LIN {X 0,Y 425.385,Z 150.495,A -85,B 0,C 180,E1 -9729.51,E2 -9729.51} C_VEL
LIN {X 0,Y 425.388,Z 150.493,A -85,B 0,C 180,E1 -9732.898,E2 -9732.898} C_VEL
LIN {X 0,Y 425.316,Z 150.502,A -85,B 0,C 180,E1 -9736.582,E2 -9736.582} C_VEL
LIN {X 0,Y 425.295,Z 150.511,A -85,B 0,C 180,E1 -9739.621,E2 -9739.621} C_VEL
LIN {X 0,Y 425.287,Z 150.506,A -85,B 0,C 180,E1 -9742.339,E2 -9742.339} C_VEL
LIN {X 0,Y 425.254,Z 150.515,A -85,B 0,C 180,E1 -9745.448,E2 -9745.448} C_VEL
LIN {X 0,Y 425.298,Z 150.505,A -85,B 0,C 180,E1 -9748.857,E2 -9748.857} C_VEL
LIN {X 0,Y 425.248,Z 150.512,A -85,B 0,C 180,E1 -9751.928,E2 -9751.928} C_VEL
LIN {X 0,Y 425.293,Z 150.512,A -85,B 0,C 180,E1 -9755.337,E2 -9755.337} C_VEL
LIN {X 0,Y 425.276,Z 150.51,A -85,B 0,C 180,E1 -9758.901,E2 -9758.901} C_VEL
LIN {X 0,Y 425.266,Z 150.508,A -85,B 0,C 180,E1 -9761.954,E2 -9761.954} C_VEL
LIN {X 0,Y 425.287,Z 150.51,A -85,B 0,C 180,E1 -9765.283,E2 -9765.283} C_VEL
LIN {X 0,Y 425.248,Z 150.513,A -85,B 0,C 180,E1 -9768.618,E2 -9768.618} C_VEL
LIN {X 0,Y 425.275,Z 150.512,A -85,B 0,C 180,E1 -9771.098,E2 -9771.098} C_VEL
LIN {X 0,Y 425.291,Z 150.51,A -85,B 0,C 180,E1 -9774.663,E2 -9774.663} C_VEL
LIN {X 0,Y 425.247,Z 150.511,A -85,B 0,C 180,E1 -9778.071,E2 -9778.071} C_VEL
LIN {X 0,Y 425.293,Z 150.509,A -85,B 0,C 180,E1 -9781.365,E2 -9781.365} C_VEL
LIN {X 0,Y 425.286,Z 150.616,A -85,B 0,C 180,E1 -9783.067,E2 -9783.067} C_VEL
LIN {X 0,Y 427.741,Z 162.985,A -85,B 0,C 180,E1 -9785.747,E2 -9785.747} C_VEL
LIN {X 0,Y 428.031,Z 166.812,A -85,B 0,C 180,E1 -9786.536,E2 -9786.536} C_VEL
LIN {X 0,Y 426.978,Z 184.548,A -85,B 0,C 180,E1 -9790.029,E2 -9790.029} C_VEL
LIN {X 0,Y 426.558,Z 191.651,A -85,B 0,C 180,E1 -9791.365,E2 -9791.365} C_VEL
LIN {X 0,Y 430.283,Z 215.837,A -85,B 0,C 180,E1 -9791.95,E2 -9791.95} C_VEL
LIN {X 0,Y 429.369,Z 299.846,A -85,B 0,C 180,E1 -9793.416,E2 -9793.416} C_VEL
LIN {X 0,Y 428.925,Z 312.927,A -85,B 0,C 180,E1 -9793.826,E2 -9793.826} C_VEL
LIN {X 0,Y 428.289,Z 325.582,A -85,B 0,C 180,E1 -9794.413,E2 -9794.413} C_VEL
LIN {X 0,Y 427.669,Z 336.858,A -85,B 0,C 180,E1 -9795.121,E2 -9795.121} C_VEL
LIN {X 0,Y 426.966,Z 348.067,A -85,B 0,C 180,E1 -9796.027,E2 -9796.027} C_VEL
LIN {X 0,Y 426.286,Z 359.035,A -85,B 0,C 180,E1 -9797.14,E2 -9797.14} C_VEL
LIN {X 0,Y 425.729,Z 368.489,A -85,B 0,C 180,E1 -9798.333,E2 -9798.333} C_VEL
LIN {X 0,Y 425.068,Z 377.599,A -85,B 0,C 180,E1 -9799.762,E2 -9799.762} C_VEL
LIN {X 0,Y 424.684,Z 384.943,A -85,B 0,C 180,E1 -9801.195,E2 -9801.195} C_VEL
LIN {X 0,Y 424.409,Z 389.909,A -85,B 0,C 180,E1 -9802.387,E2 -9802.387} C_VEL
LIN {X 0,Y 424.215,Z 394.477,A -85,B 0,C 180,E1 -9803.734,E2 -9803.734} C_VEL
LIN {X 0,Y 424.197,Z 398.42,A -85,B 0,C 180,E1 -9805.248,E2 -9805.248} C_VEL
LIN {X 0,Y 424.097,Z 400.322,A -85,B 0,C 180,E1 -9806.199,E2 -9806.199} C_VEL
LIN {X 0,Y 424.131,Z 401.769,A -85,B 0,C 180,E1 -9807.151,E2 -9807.151} C_VEL
LIN {X 0,Y 424.129,Z 402.789,A -85,B 0,C 180,E1 -9808.101,E2 -9808.101} C_VEL
LIN {X 0,Y 424.086,Z 403.653,A -85,B 0,C 180,E1 -9810,E2 -9810} C_VEL
LIN {X 0,Y 424.089,Z 403.462,A -85,B 0,C 180,E1 -9810.95,E2 -9810.95} C_VEL
LIN {X 0,Y 424.129,Z 402.861,A -85,B 0,C 180,E1 -9811.899,E2 -9811.899} C_VEL
LIN {X 0,Y 424.131,Z 401.868,A -85,B 0,C 180,E1 -9812.849,E2 -9812.849} C_VEL
LIN {X 0,Y 424.097,Z 400.476,A -85,B 0,C 180,E1 -9813.801,E2 -9813.801} C_VEL
LIN {X 0,Y 424.203,Z 397.541,A -85,B 0,C 180,E1 -9815.228,E2 -9815.228} C_VEL
LIN {X 0,Y 424.3,Z 393.567,A -85,B 0,C 180,E1 -9816.658,E2 -9816.658} C_VEL
LIN {X 0,Y 424.579,Z 387.467,A -85,B 0,C 180,E1 -9818.328,E2 -9818.328} C_VEL
LIN {X 0,Y 424.937,Z 380.79,A -85,B 0,C 180,E1 -9819.76,E2 -9819.76} C_VEL
LIN {X 0,Y 425.457,Z 372.508,A -85,B 0,C 180,E1 -9821.192,E2 -9821.192} C_VEL
LIN {X 0,Y 426.154,Z 364.041,A -85,B 0,C 180,E1 -9822.38,E2 -9822.38} C_VEL
LIN {X 0,Y 426.763,Z 354.107,A -85,B 0,C 180,E1 -9823.519,E2 -9823.519} C_VEL
LIN {X 0,Y 427.468,Z 343.265,A -85,B 0,C 180,E1 -9824.521,E2 -9824.521} C_VEL
LIN {X 0,Y 428.174,Z 331.977,A -85,B 0,C 180,E1 -9825.348,E2 -9825.348} C_VEL
LIN {X 0,Y 428.86,Z 320.52,A -85,B 0,C 180,E1 -9825.993,E2 -9825.993} C_VEL
LIN {X 0,Y 429.422,Z 307.452,A -85,B 0,C 180,E1 -9826.521,E2 -9826.521} C_VEL
LIN {X 0,Y 429.866,Z 295.022,A -85,B 0,C 180,E1 -9826.839,E2 -9826.839} C_VEL
LIN {X 0,Y 430.583,Z 214.639,A -85,B 0,C 180,E1 -9828.243,E2 -9828.243} C_VEL
LIN {X 0,Y 426.663,Z 190.71,A -85,B 0,C 180,E1 -9828.874,E2 -9828.874} C_VEL
LIN {X 0,Y 427.697,Z 173.58,A -85,B 0,C 180,E1 -9832.206,E2 -9832.206} C_VEL
LIN {X 0,Y 428.096,Z 164.652,A -85,B 0,C 180,E1 -9833.974,E2 -9833.974} C_VEL
LIN {X 0,Y 426.1,Z 154.421,A -85,B 0,C 180,E1 -9836.181,E2 -9836.181} C_VEL
LIN {X 0,Y 425.257,Z 150.515,A -85,B 0,C 180,E1 -9837.094,E2 -9837.094} C_VEL
LIN {X 0,Y 425.272,Z 150.518,A -85,B 0,C 180,E1 -9839.721,E2 -9839.721} C_VEL
LIN {X 0,Y 425.261,Z 150.519,A -85,B 0,C 180,E1 -9843.05,E2 -9843.05} C_VEL
LIN {X 0,Y 425.275,Z 150.509,A -85,B 0,C 180,E1 -9845.927,E2 -9845.927} C_VEL
LIN {X 0,Y 425.245,Z 150.519,A -85,B 0,C 180,E1 -9849.034,E2 -9849.034} C_VEL
LIN {X 0,Y 425.256,Z 150.513,A -85,B 0,C 180,E1 -9852.656,E2 -9852.656} C_VEL
LIN {X 0,Y 425.286,Z 150.513,A -85,B 0,C 180,E1 -9855.283,E2 -9855.283} C_VEL
LIN {X 0,Y 425.246,Z 150.515,A -85,B 0,C 180,E1 -9858.618,E2 -9858.618} C_VEL
LIN {X 0,Y 425.27,Z 150.51,A -85,B 0,C 180,E1 -9862.305,E2 -9862.305} C_VEL
LIN {X 0,Y 425.285,Z 150.506,A -85,B 0,C 180,E1 -9865.815,E2 -9865.815} C_VEL
LIN {X 0,Y 425.287,Z 150.507,A -85,B 0,C 180,E1 -9869.241,E2 -9869.241} C_VEL
LIN {X 0,Y 425.24,Z 150.513,A -85,B 0,C 180,E1 -9872.435,E2 -9872.435} C_VEL
LIN {X 0,Y 425.315,Z 150.498,A -85,B 0,C 180,E1 -9875.6,E2 -9875.6} C_VEL
LIN {X 0,Y 425.275,Z 150.506,A -85,B 0,C 180,E1 -9878.681,E2 -9878.681} C_VEL
LIN {X 0,Y 425.283,Z 150.507,A -85,B 0,C 180,E1 -9881.7,E2 -9881.7} C_VEL
LIN {X 0,Y 425.281,Z 150.506,A -85,B 0,C 180,E1 -9884.668,E2 -9884.668} C_VEL
LIN {X 0,Y 425.404,Z 150.491,A -85,B 0,C 180,E1 -9887.598,E2 -9887.598} C_VEL
LIN {X 0,Y 425.398,Z 150.491,A -85,B 0,C 180,E1 -9891.449,E2 -9891.449} C_VEL
LIN {X 0,Y 425.509,Z 150.478,A -85,B 0,C 180,E1 -9894.313,E2 -9894.313} C_VEL
LIN {X 0,Y 425.568,Z 150.469,A -85,B 0,C 180,E1 -9898.107,E2 -9898.107} C_VEL
LIN {X 0,Y 425.576,Z 150.474,A -85,B 0,C 180,E1 -9900,E2 -9900} C_VEL
LIN {X 0,Y 425.515,Z 150.477,A -85,B 0,C 180,E1 -9902.84,E2 -9902.84} C_VEL
LIN {X 0,Y 425.48,Z 150.483,A -85,B 0,C 180,E1 -9906.64,E2 -9906.64} C_VEL
LIN {X 0,Y 425.385,Z 150.494,A -85,B 0,C 180,E1 -9909.51,E2 -9909.51} C_VEL
LIN {X 0,Y 425.397,Z 150.491,A -85,B 0,C 180,E1 -9912.903,E2 -9912.903} C_VEL
LIN {X 0,Y 425.317,Z 150.504,A -85,B 0,C 180,E1 -9916.583,E2 -9916.583} C_VEL
LIN {X 0,Y 425.3,Z 150.511,A -85,B 0,C 180,E1 -9919.623,E2 -9919.623} C_VEL
LIN {X 0,Y 425.29,Z 150.508,A -85,B 0,C 180,E1 -9922.339,E2 -9922.339} C_VEL
LIN {X 0,Y 425.263,Z 150.517,A -85,B 0,C 180,E1 -9925.448,E2 -9925.448} C_VEL
LIN {X 0,Y 425.303,Z 150.508,A -85,B 0,C 180,E1 -9928.858,E2 -9928.858} C_VEL
LIN {X 0,Y 425.265,Z 150.515,A -85,B 0,C 180,E1 -9931.927,E2 -9931.927} C_VEL
LIN {X 0,Y 425.334,Z 150.596,A -85,B 0,C 180,E1 -9934.904,E2 -9934.904} C_VEL
LIN {X 0,Y 427.235,Z 160.421,A -85,B 0,C 180,E1 -9937.196,E2 -9937.196} C_VEL
LIN {X 0,Y 427.18,Z 167.317,A -85,B 0,C 180,E1 -9938.696,E2 -9938.696} C_VEL
LIN {X 0,Y 427.085,Z 169.637,A -85,B 0,C 180,E1 -9939.194,E2 -9939.194} C_VEL
LIN {X 0,Y 430.988,Z 189.046,A -85,B 0,C 180,E1 -9939.754,E2 -9939.754} C_VEL
LIN {X 0,Y 429.823,Z 277.143,A -85,B 0,C 180,E1 -9941.297,E2 -9941.297} C_VEL
LIN {X 0,Y 429.424,Z 290.591,A -85,B 0,C 180,E1 -9941.725,E2 -9941.725} C_VEL
LIN {X 0,Y 429.039,Z 302.325,A -85,B 0,C 180,E1 -9942.279,E2 -9942.279} C_VEL
LIN {X 0,Y 428.363,Z 314.074,A -85,B 0,C 180,E1 -9943.013,E2 -9943.013} C_VEL
LIN {X 0,Y 427.692,Z 324.645,A -85,B 0,C 180,E1 -9943.865,E2 -9943.865} C_VEL
LIN {X 0,Y 427.001,Z 335.376,A -85,B 0,C 180,E1 -9944.948,E2 -9944.948} C_VEL
LIN {X 0,Y 426.325,Z 345.223,A -85,B 0,C 180,E1 -9946.181,E2 -9946.181} C_VEL
LIN {X 0,Y 425.719,Z 353.142,A -85,B 0,C 180,E1 -9947.402,E2 -9947.402} C_VEL
LIN {X 0,Y 425.175,Z 360.816,A -85,B 0,C 180,E1 -9948.864,E2 -9948.864} C_VEL
LIN {X 0,Y 424.74,Z 367.339,A -85,B 0,C 180,E1 -9950.428,E2 -9950.428} C_VEL
LIN {X 0,Y 424.409,Z 372.967,A -85,B 0,C 180,E1 -9952.214,E2 -9952.214} C_VEL
LIN {X 0,Y 424.279,Z 375.771,A -85,B 0,C 180,E1 -9953.392,E2 -9953.392} C_VEL
LIN {X 0,Y 424.1,Z 377.826,A -85,B 0,C 180,E1 -9954.549,E2 -9954.549} C_VEL
LIN {X 0,Y 423.961,Z 379.542,A -85,B 0,C 180,E1 -9955.981,E2 -9955.981} C_VEL
LIN {X 0,Y 423.947,Z 380.391,A -85,B 0,C 180,E1 -9957.721,E2 -9957.721} C_VEL
LIN {X 0,Y 423.986,Z 379.875,A -85,B 0,C 180,E1 -9959.537,E2 -9959.537} C_VEL
LIN {X 0,Y 424.112,Z 377.719,A -85,B 0,C 180,E1 -9961.435,E2 -9961.435} C_VEL
LIN {X 0,Y 424.305,Z 374.922,A -85,B 0,C 180,E1 -9962.903,E2 -9962.903} C_VEL
LIN {X 0,Y 424.55,Z 370.642,A -85,B 0,C 180,E1 -9964.507,E2 -9964.507} C_VEL
LIN {X 0,Y 424.777,Z 365.04,A -85,B 0,C 180,E1 -9966.086,E2 -9966.086} C_VEL
LIN {X 0,Y 425.245,Z 357.799,A -85,B 0,C 180,E1 -9967.659,E2 -9967.659} C_VEL
LIN {X 0,Y 425.74,Z 350.363,A -85,B 0,C 180,E1 -9968.958,E2 -9968.958} C_VEL
LIN {X 0,Y 426.309,Z 342.255,A -85,B 0,C 180,E1 -9970.124,E2 -9970.124} C_VEL
LIN {X 0,Y 426.924,Z 332.513,A -85,B 0,C 180,E1 -9971.276,E2 -9971.276} C_VEL
LIN {X 0,Y 427.64,Z 322.198,A -85,B 0,C 180,E1 -9972.254,E2 -9972.254} C_VEL
LIN {X 0,Y 428.262,Z 309.768,A -85,B 0,C 180,E1 -9973.188,E2 -9973.188} C_VEL
LIN {X 0,Y 428.803,Z 297.552,A -85,B 0,C 180,E1 -9973.883,E2 -9973.883} C_VEL
LIN {X 0,Y 429.235,Z 285.099,A -85,B 0,C 180,E1 -9974.387,E2 -9974.387} C_VEL
LIN {X 0,Y 429.463,Z 276.095,A -85,B 0,C 180,E1 -9974.643,E2 -9974.643} C_VEL
LIN {X 0,Y 428.945,Z 270.305,A -85,B 0,C 180,E1 -9974.782,E2 -9974.782} C_VEL
LIN {X 0,Y 423.695,Z 251.592,A -85,B 0,C 180,E1 -9975.317,E2 -9975.317} C_VEL
LIN {X 0,Y 423.075,Z 245.782,A -85,B 0,C 180,E1 -9975.443,E2 -9975.443} C_VEL
LIN {X 0,Y 423.731,Z 189.379,A -85,B 0,C 180,E1 -9976.431,E2 -9976.431} C_VEL
LIN {X 0,Y 419.899,Z 169.602,A -85,B 0,C 180,E1 -9976.972,E2 -9976.972} C_VEL
LIN {X 0,Y 420.164,Z 161.037,A -85,B 0,C 180,E1 -9978.909,E2 -9978.909} C_VEL
LIN {X 0,Y 418.398,Z 151.37,A -85,B 0,C 180,E1 -9981.274,E2 -9981.274} C_VEL
LIN {X 0,Y 418.49,Z 151.358,A -85,B 0,C 180,E1 -9984.217,E2 -9984.217} C_VEL
LIN {X 0,Y 418.543,Z 151.349,A -85,B 0,C 180,E1 -9988.075,E2 -9988.075} C_VEL
LIN {X 0,Y 418.475,Z 151.355,A -85,B 0,C 180,E1 -9990.962,E2 -9990.962} C_VEL
LIN {X 0,Y 418.475,Z 151.355,A -85,B 0,C 180,E1 -9992.888,E2 -9992.888} C_VEL
LIN {X 0,Y 418.487,Z 151.355,A -85,B 0,C 180,E1 -9995.783,E2 -9995.783} C_VEL
LIN {X 0,Y 418.379,Z 151.368,A -85,B 0,C 180,E1 -9998.696,E2 -9998.696} C_VEL
LIN {X 0,Y 418.316,Z 151.376,A -85,B 0,C 180,E1 -10001.631,E2 -10001.631} C_VEL
LIN {X 0,Y 418.281,Z 151.379,A -85,B 0,C 180,E1 -10004.598,E2 -10004.598} C_VEL
LIN {X 0,Y 418.258,Z 151.384,A -85,B 0,C 180,E1 -10007.605,E2 -10007.605} C_VEL
LIN {X 0,Y 418.252,Z 151.382,A -85,B 0,C 180,E1 -10010.663,E2 -10010.663} C_VEL
LIN {X 0,Y 418.261,Z 151.388,A -85,B 0,C 180,E1 -10013.783,E2 -10013.783} C_VEL
LIN {X 0,Y 418.211,Z 151.388,A -85,B 0,C 180,E1 -10017.043,E2 -10017.043} C_VEL
LIN {X 0,Y 418.244,Z 151.384,A -85,B 0,C 180,E1 -10020.272,E2 -10020.272} C_VEL
LIN {X 0,Y 418.235,Z 151.39,A -85,B 0,C 180,E1 -10023.679,E2 -10023.679} C_VEL
LIN {X 0,Y 418.241,Z 151.387,A -85,B 0,C 180,E1 -10027.224,E2 -10027.224} C_VEL
LIN {X 0,Y 418.209,Z 151.389,A -85,B 0,C 180,E1 -10030.867,E2 -10030.867} C_VEL
LIN {X 0,Y 418.205,Z 151.39,A -85,B 0,C 180,E1 -10033.728,E2 -10033.728} C_VEL
LIN {X 0,Y 418.202,Z 151.388,A -85,B 0,C 180,E1 -10036.447,E2 -10036.447} C_VEL
LIN {X 0,Y 418.213,Z 151.393,A -85,B 0,C 180,E1 -10039.132,E2 -10039.132} C_VEL
LIN {X 0,Y 418.241,Z 151.386,A -85,B 0,C 180,E1 -10042.776,E2 -10042.776} C_VEL
LIN {X 0,Y 418.236,Z 151.384,A -85,B 0,C 180,E1 -10046.321,E2 -10046.321} C_VEL
LIN {X 0,Y 418.242,Z 151.383,A -85,B 0,C 180,E1 -10049.728,E2 -10049.728} C_VEL
LIN {X 0,Y 418.224,Z 151.39,A -85,B 0,C 180,E1 -10053.017,E2 -10053.017} C_VEL
LIN {X 0,Y 418.262,Z 151.382,A -85,B 0,C 180,E1 -10056.217,E2 -10056.217} C_VEL
LIN {X 0,Y 418.251,Z 151.383,A -85,B 0,C 180,E1 -10059.337,E2 -10059.337} C_VEL
LIN {X 0,Y 418.259,Z 151.385,A -85,B 0,C 180,E1 -10062.395,E2 -10062.395} C_VEL
LIN {X 0,Y 418.28,Z 151.378,A -85,B 0,C 180,E1 -10065.402,E2 -10065.402} C_VEL
LIN {X 0,Y 418.317,Z 151.38,A -85,B 0,C 180,E1 -10068.369,E2 -10068.369} C_VEL
LIN {X 0,Y 418.45,Z 151.363,A -85,B 0,C 180,E1 -10072.278,E2 -10072.278} C_VEL
LIN {X 0,Y 418.487,Z 151.358,A -85,B 0,C 180,E1 -10074.217,E2 -10074.217} C_VEL
LIN {X 0,Y 418.538,Z 151.351,A -85,B 0,C 180,E1 -10078.075,E2 -10078.075} C_VEL
LIN {X 0,Y 418.411,Z 151.362,A -85,B 0,C 180,E1 -10080.962,E2 -10080.962} C_VEL
LIN {X 0,Y 418.472,Z 151.355,A -85,B 0,C 180,E1 -10082.888,E2 -10082.888} C_VEL
LIN {X 0,Y 418.473,Z 151.358,A -85,B 0,C 180,E1 -10085.783,E2 -10085.783} C_VEL
LIN {X 0,Y 418.37,Z 151.368,A -85,B 0,C 180,E1 -10088.696,E2 -10088.696} C_VEL
LIN {X 0,Y 418.304,Z 151.379,A -85,B 0,C 180,E1 -10091.631,E2 -10091.631} C_VEL
LIN {X 0,Y 418.28,Z 151.382,A -85,B 0,C 180,E1 -10093.605,E2 -10093.605} C_VEL
LIN {X 0,Y 418.255,Z 151.381,A -85,B 0,C 180,E1 -10096.707,E2 -10096.707} C_VEL
LIN {X 0,Y 418.239,Z 151.39,A -85,B 0,C 180,E1 -10099.777,E2 -10099.777} C_VEL
LIN {X 0,Y 418.227,Z 151.385,A -85,B 0,C 180,E1 -10102.737,E2 -10102.737} C_VEL
LIN {X 0,Y 418.213,Z 151.39,A -85,B 0,C 180,E1 -10105.908,E2 -10105.908} C_VEL
LIN {X 0,Y 418.257,Z 151.385,A -85,B 0,C 180,E1 -10109.163,E2 -10109.163} C_VEL
LIN {X 0,Y 418.233,Z 151.384,A -85,B 0,C 180,E1 -10112.529,E2 -10112.529} C_VEL
LIN {X 0,Y 418.25,Z 151.384,A -85,B 0,C 180,E1 -10114.842,E2 -10114.842} C_VEL
LIN {X 0,Y 418.234,Z 151.384,A -85,B 0,C 180,E1 -10118.444,E2 -10118.444} C_VEL
LIN {X 0,Y 418.22,Z 151.386,A -85,B 0,C 180,E1 -10122.236,E2 -10122.236} C_VEL
LIN {X 0,Y 418.238,Z 151.391,A -85,B 0,C 180,E1 -10125.108,E2 -10125.108} C_VEL
LIN {X 0,Y 418.219,Z 151.386,A -85,B 0,C 180,E1 -10127.764,E2 -10127.764} C_VEL
LIN {X 0,Y 418.233,Z 151.385,A -85,B 0,C 180,E1 -10131.556,E2 -10131.556} C_VEL
LIN {X 0,Y 418.249,Z 151.386,A -85,B 0,C 180,E1 -10135.158,E2 -10135.158} C_VEL
LIN {X 0,Y 418.232,Z 151.385,A -85,B 0,C 180,E1 -10137.47,E2 -10137.47} C_VEL
LIN {X 0,Y 418.258,Z 151.388,A -85,B 0,C 180,E1 -10140.898,E2 -10140.898} C_VEL
LIN {X 0,Y 418.244,Z 151.543,A -85,B 0,C 180,E1 -10142.836,E2 -10142.836} C_VEL
LIN {X 0,Y 420.739,Z 163.972,A -85,B 0,C 180,E1 -10145.58,E2 -10145.58} C_VEL
LIN {X 0,Y 421.099,Z 167.806,A -85,B 0,C 180,E1 -10146.387,E2 -10146.387} C_VEL
LIN {X 0,Y 419.984,Z 185.789,A -85,B 0,C 180,E1 -10149.988,E2 -10149.988} C_VEL
LIN {X 0,Y 419.56,Z 191.228,A -85,B 0,C 180,E1 -10151.057,E2 -10151.057} C_VEL
LIN {X 0,Y 423.488,Z 216.496,A -85,B 0,C 180,E1 -10151.684,E2 -10151.684} C_VEL
LIN {X 0,Y 422.529,Z 300.028,A -85,B 0,C 180,E1 -10153.171,E2 -10153.171} C_VEL
LIN {X 0,Y 422,Z 313.739,A -85,B 0,C 180,E1 -10153.616,E2 -10153.616} C_VEL
LIN {X 0,Y 421.371,Z 326.109,A -85,B 0,C 180,E1 -10154.212,E2 -10154.212} C_VEL
LIN {X 0,Y 420.684,Z 337.985,A -85,B 0,C 180,E1 -10154.992,E2 -10154.992} C_VEL
LIN {X 0,Y 419.928,Z 349.864,A -85,B 0,C 180,E1 -10155.998,E2 -10155.998} C_VEL
LIN {X 0,Y 419.252,Z 359.727,A -85,B 0,C 180,E1 -10157.044,E2 -10157.044} C_VEL
LIN {X 0,Y 418.588,Z 369.804,A -85,B 0,C 180,E1 -10158.377,E2 -10158.377} C_VEL
LIN {X 0,Y 417.988,Z 378.668,A -85,B 0,C 180,E1 -10159.831,E2 -10159.831} C_VEL
LIN {X 0,Y 417.566,Z 385.75,A -85,B 0,C 180,E1 -10161.287,E2 -10161.287} C_VEL
LIN {X 0,Y 417.271,Z 391.405,A -85,B 0,C 180,E1 -10162.743,E2 -10162.743} C_VEL
LIN {X 0,Y 417.097,Z 395.847,A -85,B 0,C 180,E1 -10164.198,E2 -10164.198} C_VEL
LIN {X 0,Y 417.104,Z 398.192,A -85,B 0,C 180,E1 -10165.167,E2 -10165.167} C_VEL
LIN {X 0,Y 417.013,Z 400.1,A -85,B 0,C 180,E1 -10166.135,E2 -10166.135} C_VEL
LIN {X 0,Y 417.028,Z 401.557,A -85,B 0,C 180,E1 -10167.102,E2 -10167.102} C_VEL
LIN {X 0,Y 417.056,Z 402.583,A -85,B 0,C 180,E1 -10168.069,E2 -10168.069} C_VEL
LIN {X 0,Y 417.006,Z 403.456,A -85,B 0,C 180,E1 -10170,E2 -10170} C_VEL
LIN {X 0,Y 417.011,Z 403.274,A -85,B 0,C 180,E1 -10170.966,E2 -10170.966} C_VEL
LIN {X 0,Y 417.056,Z 402.677,A -85,B 0,C 180,E1 -10171.931,E2 -10171.931} C_VEL
LIN {X 0,Y 417.027,Z 401.688,A -85,B 0,C 180,E1 -10172.898,E2 -10172.898} C_VEL
LIN {X 0,Y 417.013,Z 400.301,A -85,B 0,C 180,E1 -10173.865,E2 -10173.865} C_VEL
LIN {X 0,Y 417.117,Z 397.375,A -85,B 0,C 180,E1 -10175.317,E2 -10175.317} C_VEL
LIN {X 0,Y 417.233,Z 393.411,A -85,B 0,C 180,E1 -10176.772,E2 -10176.772} C_VEL
LIN {X 0,Y 417.52,Z 387.326,A -85,B 0,C 180,E1 -10178.47,E2 -10178.47} C_VEL
LIN {X 0,Y 417.919,Z 380.659,A -85,B 0,C 180,E1 -10179.926,E2 -10179.926} C_VEL
LIN {X 0,Y 418.482,Z 372.388,A -85,B 0,C 180,E1 -10181.381,E2 -10181.381} C_VEL
LIN {X 0,Y 419.21,Z 363.938,A -85,B 0,C 180,E1 -10182.588,E2 -10182.588} C_VEL
LIN {X 0,Y 419.869,Z 353.613,A -85,B 0,C 180,E1 -10183.789,E2 -10183.789} C_VEL
LIN {X 0,Y 420.694,Z 341.782,A -85,B 0,C 180,E1 -10184.883,E2 -10184.883} C_VEL
LIN {X 0,Y 421.434,Z 330.112,A -85,B 0,C 180,E1 -10185.723,E2 -10185.723} C_VEL
LIN {X 0,Y 422.189,Z 318.017,A -85,B 0,C 180,E1 -10186.377,E2 -10186.377} C_VEL
LIN {X 0,Y 422.731,Z 305.823,A -85,B 0,C 180,E1 -10186.852,E2 -10186.852} C_VEL
LIN {X 0,Y 423.104,Z 292.419,A -85,B 0,C 180,E1 -10187.179,E2 -10187.179} C_VEL
LIN {X 0,Y 423.908,Z 215.634,A -85,B 0,C 180,E1 -10188.538,E2 -10188.538} C_VEL
LIN {X 0,Y 419.745,Z 190.559,A -85,B 0,C 180,E1 -10189.207,E2 -10189.207} C_VEL
LIN {X 0,Y 420.759,Z 174.753,A -85,B 0,C 180,E1 -10192.334,E2 -10192.334} C_VEL
LIN {X 0,Y 421.259,Z 167.111,A -85,B 0,C 180,E1 -10193.864,E2 -10193.864} C_VEL
LIN {X 0,Y 419.416,Z 156.904,A -85,B 0,C 180,E1 -10196.095,E2 -10196.095} C_VEL
LIN {X 0,Y 418.192,Z 151.395,A -85,B 0,C 180,E1 -10197.377,E2 -10197.377} C_VEL
LIN {X 0,Y 418.235,Z 151.392,A -85,B 0,C 180,E1 -10200.273,E2 -10200.273} C_VEL
LIN {X 0,Y 418.228,Z 151.392,A -85,B 0,C 180,E1 -10203.679,E2 -10203.679} C_VEL
LIN {X 0,Y 418.232,Z 151.391,A -85,B 0,C 180,E1 -10207.225,E2 -10207.225} C_VEL
LIN {X 0,Y 418.207,Z 151.396,A -85,B 0,C 180,E1 -10210.95,E2 -10210.95} C_VEL
LIN {X 0,Y 418.202,Z 151.391,A -85,B 0,C 180,E1 -10213.728,E2 -10213.728} C_VEL
LIN {X 0,Y 418.2,Z 151.393,A -85,B 0,C 180,E1 -10216.447,E2 -10216.447} C_VEL
LIN {X 0,Y 418.207,Z 151.391,A -85,B 0,C 180,E1 -10219.133,E2 -10219.133} C_VEL
LIN {X 0,Y 418.233,Z 151.387,A -85,B 0,C 180,E1 -10222.775,E2 -10222.775} C_VEL
LIN {X 0,Y 418.229,Z 151.387,A -85,B 0,C 180,E1 -10226.321,E2 -10226.321} C_VEL
LIN {X 0,Y 418.236,Z 151.383,A -85,B 0,C 180,E1 -10229.727,E2 -10229.727} C_VEL
LIN {X 0,Y 418.204,Z 151.391,A -85,B 0,C 180,E1 -10233.016,E2 -10233.016} C_VEL
LIN {X 0,Y 418.226,Z 151.384,A -85,B 0,C 180,E1 -10236.215,E2 -10236.215} C_VEL
LIN {X 0,Y 418.231,Z 151.378,A -85,B 0,C 180,E1 -10239.336,E2 -10239.336} C_VEL
LIN {X 0,Y 418.237,Z 151.39,A -85,B 0,C 180,E1 -10242.394,E2 -10242.394} C_VEL
LIN {X 0,Y 418.253,Z 151.38,A -85,B 0,C 180,E1 -10245.401,E2 -10245.401} C_VEL
LIN {X 0,Y 418.349,Z 151.37,A -85,B 0,C 180,E1 -10247.385,E2 -10247.385} C_VEL
LIN {X 0,Y 418.323,Z 151.375,A -85,B 0,C 180,E1 -10250.328,E2 -10250.328} C_VEL
LIN {X 0,Y 418.442,Z 151.351,A -85,B 0,C 180,E1 -10253.248,E2 -10253.248} C_VEL
LIN {X 0,Y 418.315,Z 151.373,A -85,B 0,C 180,E1 -10255.181,E2 -10255.181} C_VEL
LIN {X 0,Y 418.537,Z 151.344,A -85,B 0,C 180,E1 -10258.075,E2 -10258.075} C_VEL
LIN {X 0,Y 418.411,Z 151.36,A -85,B 0,C 180,E1 -10260.962,E2 -10260.962} C_VEL
LIN {X 0,Y 418.472,Z 151.354,A -85,B 0,C 180,E1 -10262.888,E2 -10262.888} C_VEL
LIN {X 0,Y 418.441,Z 151.358,A -85,B 0,C 180,E1 -10266.491,E2 -10266.491} C_VEL
LIN {X 0,Y 418.371,Z 151.366,A -85,B 0,C 180,E1 -10268.696,E2 -10268.696} C_VEL
LIN {X 0,Y 418.358,Z 151.368,A -85,B 0,C 180,E1 -10272.614,E2 -10272.614} C_VEL
LIN {X 0,Y 418.253,Z 151.385,A -85,B 0,C 180,E1 -10275.596,E2 -10275.596} C_VEL
LIN {X 0,Y 418.241,Z 151.385,A -85,B 0,C 180,E1 -10278.619,E2 -10278.619} C_VEL
LIN {X 0,Y 418.231,Z 151.392,A -85,B 0,C 180,E1 -10281.697,E2 -10281.697} C_VEL
